(* CoDeSys 2.3.9.41 project: KS Sheksninskaya.pro *)
(* Libraries: PID_Regulators.lib 6.11.19 15:29:27, Util.lib 18.5.10 15:14:28, Germes_1_0.lib 3.5.20 13:44:14, STANDARD.LIB 4.10.05 11:14:46, IECSFC.LIB 13.4.06 15:51:28, SYSLIBTIME.LIB 6.11.19 15:29:28, ANALYZATION.LIB 5.10.99 09:05:06 *)

(* PLC configuration (modules and I/O channels)
Fast discrete inputs [I_SIMPLE_INPUT] node 0, in %IB0 out %QB0 {Filtrationtime = 10}
  DD2_7_DI0 AT %IX0.0 [BitInput] Импульсный счетчик FQS03.01
  DD2_7_DI1 AT %IX0.1 [BitInput] резерв
  DD2_7_DI2 AT %IX0.2 [BitInput] резерв
  DD2_7_DI3 AT %IX0.3 [BitInput] резерв
Discrete inputs [ID130] node 1, in %IB1 out %QB1 {Filtrationtime_GeneralINP = 10; Visibility = No; PinCount = 12}
  AT %IB1.0 [ByteInput] 8 discrete inputs
  AT %IB1.1 [ByteInput] 4 discrete inputs
Discrete outputs [ID131] node 2, in %IB2 out %QB2 {SafeValueByte = 0; SafeValueByteM = 0; Visibility = No; PinCount = 12}
  AT %QB2.0 [ByteOutput] 8 discrete outputs
  AT %QB2.1 [ByteOutput] 4 discrete outputs
Fast analog inputs [ID125] node 3, in %IB3 out %QB3 {Flt_Comm = 50Hz 2Por}
  DD2_7_AI0 AT %IR3.0 [FloatInputP] Датчик температуры в помещении {AIN_TYPE = 0-20 mA; Peak_Filtr = 200; Flt_Ch = Off; TauRC = 10; MinFV = 0; MaxFV = 20}
  DD2_7_AI1 AT %IR3.1 [FloatInputP] Расходомер FT01.01 {AIN_TYPE = 0-20 mA; Peak_Filtr = 200; Flt_Ch = Off; TauRC = 10; MinFV = 0; MaxFV = 20}
  DD2_7_AI2 AT %IR3.2 [FloatInputP] Расходомер FT01.02 {AIN_TYPE = 0-20 mA; Peak_Filtr = 200; Flt_Ch = Off; TauRC = 10; MinFV = 0; MaxFV = 20}
  DD2_7_AI3 AT %IR3.3 [FloatInputP] рН/ОВП метр QE01.01 {AIN_TYPE = 0-20 mA; Peak_Filtr = 200; Flt_Ch = Off; TauRC = 10; MinFV = 0; MaxFV = 20}
  DD2_7_AI4 AT %IR3.4 [FloatInputP] рН/ОВП метр QE01.02 {AIN_TYPE = 0-20 mA; Peak_Filtr = 200; Flt_Ch = Off; TauRC = 10; MinFV = 0; MaxFV = 20}
  DD2_7_AI5 AT %IR3.5 [FloatInputP] Давление на входе в фильтр-пресс {AIN_TYPE = 0-20 mA; Peak_Filtr = 200; Flt_Ch = Off; TauRC = 10; MinFV = 0; MaxFV = 20}
  DD2_7_AI6 AT %IR3.6 [FloatInputP] резерв {AIN_TYPE = 0-20 mA; Peak_Filtr = 200; Flt_Ch = Off; TauRC = 10; MinFV = 0; MaxFV = 20}
  DD2_7_AI7 AT %IR3.7 [FloatInputP] резерв {AIN_TYPE = 0-20 mA; Peak_Filtr = 200; Flt_Ch = Off; TauRC = 10; MinFV = 0; MaxFV = 20}
  AT %IW3.8 [WordInput] AI read time (10ms)
Analog outputs [ID126] node 4, in %IB4 out %QB4
  DD2_7_AO0 AT %QR4.0 [FloatOutputP] Управление НД08.04 {AOUT_TYPE = 4-20 mA; SafeValueREAL = 0.0}
  DD2_7_AO1 AT %QR4.1 [FloatOutputP] резерв {AOUT_TYPE = 4-20 mA; SafeValueREAL = 0.0}
  DD2_7_AO2 AT %QR4.2 [FloatOutputP] резерв {AOUT_TYPE = 4-20 mA; SafeValueREAL = 0.0}
  DD2_7_AO3 AT %QR4.3 [FloatOutputP] резерв {AOUT_TYPE = 4-20 mA; SafeValueREAL = 0.0}
Special input [ID103] node 5, in %IB5 out %QB5 {Filtrationtime = 1000; PinCount = 1; WatchDogPeriod = 400; PollPeriod = 3000; Visibility = No}
  AT %IX5.0 [BitInput] Special input
Special output [ID104] node 6, in %IB6 out %QB6 {Visibility = No; PinCount = 1}
  AT %QX6.0 [BitOutput] Special output
ModBus (Master) [MODBUS_MASTER_ID450] node 7, in %IB7 out %QB7 {Visibility = No}
  LastAddress AT %QD7.0 [DWordOutput] Last address
  LastError AT %QW7.1 [WordOutput] Last error
  RS-485-1 [COM1_USART] node 0, in %IB7.0 out %QB7.0 {CommunicationSpeed = 9600; Parity = EVEN; BitLength = 8 bits; StopLength = One stop bit; InterfaceType = RS485; FrameOriented = RTU; Timeout = 0; Visibility = No}
  Universal Modbus device [ID2000] node 1, in %IB7.1 out %QB7.1 {ModuleIP = 10:0:0:101; ServiceTimeout = 20; TCPport = 502; NetMode = Serial; ModuleSlaveAddress = 11; RequestType = Both; PeriodOfService = 100; Visibility = No; RepeatCounter = 0; ByteSequence = Trace_mode}
    AT %QB7.1.0 [ComChannel] Command (0xff - Start)
    32bit output module [ID2006] node 0, in %IB7.1.0 out %QB7.1.0 {ModbusAddress = 0; Command_write_regs = Force multiple coils (0x0f); Visibility = No}
      DD1_1_DO AT %QD7.1.0.0 [DWordOutput]
  Universal Modbus device [ID2000] node 2, in %IB7.2 out %QB7.2 {ModuleIP = 10:0:0:102; ServiceTimeout = 20; TCPport = 502; NetMode = Serial; ModuleSlaveAddress = 12; RequestType = By poll time; PeriodOfService = 100; Visibility = No; RepeatCounter = 0; ByteSequence = Trace_mode}
    AT %QB7.2.0 [ComChannel] Command (0xff - Start)
DD1_2_DI AT %ID7.2.0.0 [DWordInput]
Universal Modbus device [ID2000] node 3, in %IB7.3 out %QB7.3 {ModuleIP = 10:0:0:103; ServiceTimeout = 20; TCPport = 502; NetMode = Serial; ModuleSlaveAddress = 13; RequestType = By poll time; PeriodOfService = 100; Visibility = No; RepeatCounter = 0; ByteSequence = Trace_mode}
  AT %QB7.3.0 [ComChannel] Command (0xff - Start)
DD1_3_DI AT %IW7.3.0.0 [WordInput]
Universal Modbus device [ID2000] node 4, in %IB7.4 out %QB7.4 {ModuleIP = 10:0:0:104; ServiceTimeout = 20; TCPport = 502; NetMode = Serial; ModuleSlaveAddress = 14; RequestType = Both; PeriodOfService = 100; Visibility = No; RepeatCounter = 0; ByteSequence = Trace_mode}
  AT %QB7.4.0 [ComChannel] Command (0xff - Start)
  Register output module [ID2004] node 0, in %IB7.4.0 out %QB7.4.0 {ModbusAddress = 0; Command_write_one_reg = Write multiple registers(0x10); Visibility = No}
    DD1_4_AO0 AT %QW7.4.0.0 [WordOutput]
  Register output module [ID2004] node 1, in %IB7.4.1 out %QB7.4.1 {ModbusAddress = 1; Command_write_one_reg = Write multiple registers(0x10); Visibility = No}
    DD1_4_AO1 AT %QW7.4.1.0 [WordOutput]
  Register output module [ID2004] node 2, in %IB7.4.2 out %QB7.4.2 {ModbusAddress = 2; Command_write_one_reg = Write multiple registers(0x10); Visibility = No}
    DD1_4_AO2 AT %QW7.4.2.0 [WordOutput]
  Register output module [ID2004] node 3, in %IB7.4.3 out %QB7.4.3 {ModbusAddress = 3; Command_write_one_reg = Write multiple registers(0x10); Visibility = No}
    DD1_4_AO3 AT %QW7.4.3.0 [WordOutput]
  Register output module [ID2004] node 4, in %IB7.4.4 out %QB7.4.4 {ModbusAddress = 4; Command_write_one_reg = Write multiple registers(0x10); Visibility = No}
    DD1_4_AO4 AT %QW7.4.4.0 [WordOutput]
  Register output module [ID2004] node 5, in %IB7.4.5 out %QB7.4.5 {ModbusAddress = 5; Command_write_one_reg = Write multiple registers(0x10); Visibility = No}
    DD1_4_AO5 AT %QW7.4.5.0 [WordOutput]
  Register output module [ID2004] node 6, in %IB7.4.6 out %QB7.4.6 {ModbusAddress = 6; Command_write_one_reg = Write multiple registers(0x10); Visibility = No}
    DD1_4_AO6 AT %QW7.4.6.0 [WordOutput]
  Register output module [ID2004] node 7, in %IB7.4.7 out %QB7.4.7 {ModbusAddress = 7; Command_write_one_reg = Write multiple registers(0x10); Visibility = No}
    DD1_4_AO7 AT %QW7.4.7.0 [WordOutput]
  AT %QB7.5.0 [ComChannel] Command (0xff - Start)
com_wordN0105 AT %QW7.5.0.0 [WordOutput]
zad_rsN0105 AT %QW7.5.1.0 [WordOutput]
stat_wordN0105 AT %IW7.5.2.0 [WordInput]
di29N0105 AT %IW7.5.3.0 [WordInput]
Universal Modbus device [ID2000] node 6, in %IB7.6 out %QB7.6 {ModuleIP = 10:0:0:106; ServiceTimeout = 20; TCPport = 502; NetMode = Serial; ModuleSlaveAddress = 16; RequestType = By poll time; PeriodOfService = 100; Visibility = No; RepeatCounter = 0; ByteSequence = Trace_mode}
  AT %QB7.6.0 [ComChannel] Command (0xff - Start)
  Register output module [ID2004] node 0, in %IB7.6.0 out %QB7.6.0 {ModbusAddress = 49999; Command_write_one_reg = Write multiple registers(0x10); Visibility = No}
    com_wordND080301 AT %QW7.6.0.0 [WordOutput]
  Register output module [ID2004] node 1, in %IB7.6.1 out %QB7.6.1 {ModbusAddress = 50009; Command_write_one_reg = Write multiple registers(0x10); Visibility = No}
    zad_rsND080301 AT %QW7.6.1.0 [WordOutput]
  Register input module [ID2003] node 2, in %IB7.6.2 out %QB7.6.2 {ModbusAddress = 50199; Command_read_regs = Read holding Registers  (0x03); Visibility = No}
    stat_wordND080301 AT %IW7.6.2.0 [WordInput]
  Register input module [ID2003] node 3, in %IB7.6.3 out %QB7.6.3 {ModbusAddress = 16609; Command_read_regs = Read holding Registers  (0x03); Visibility = No}
    di29ND080301 AT %IW7.6.3.0 [WordInput]
Universal Modbus device [ID2000] node 7, in %IB7.7 out %QB7.7 {ModuleIP = 10:0:0:107; ServiceTimeout = 20; TCPport = 502; NetMode = Serial; ModuleSlaveAddress = 17; RequestType = By poll time; PeriodOfService = 100; Visibility = No; RepeatCounter = 0; ByteSequence = Trace_mode}
  AT %QB7.7.0 [ComChannel] Command (0xff - Start)
com_wordND080302 AT %QW7.7.0.0 [WordOutput]
zad_rsND080302 AT %QW7.7.1.0 [WordOutput]
stat_wordND080302 AT %IW7.7.2.0 [WordInput]
di29ND080302 AT %IW7.7.3.0 [WordInput]
Universal Modbus device [ID2000] node 8, in %IB7.8 out %QB7.8 {ModuleIP = 10:0:0:201; ServiceTimeout = 20; TCPport = 502; NetMode = Serial; ModuleSlaveAddress = 21; RequestType = Both; PeriodOfService = 100; Visibility = No; RepeatCounter = 0; ByteSequence = Trace_mode}
  AT %QB7.8.0 [ComChannel] Command (0xff - Start)
  32bit output module [ID2006] node 0, in %IB7.8.0 out %QB7.8.0 {ModbusAddress = 0; Command_write_regs = Force multiple coils (0x0f); Visibility = No}
    DD2_1_DO AT %QD7.8.0.0 [DWordOutput]
Universal Modbus device [ID2000] node 9, in %IB7.9 out %QB7.9 {ModuleIP = 10:0:0:202; ServiceTimeout = 20; TCPport = 502; NetMode = Serial; ModuleSlaveAddress = 22; RequestType = Both; PeriodOfService = 100; Visibility = No; RepeatCounter = 0; ByteSequence = Trace_mode}
  AT %QB7.9.0 [ComChannel] Command (0xff - Start)
DD2_2_DO AT %QD7.9.0.0 [DWordOutput]
Universal Modbus device [ID2000] node 10, in %IB7.10 out %QB7.10 {ModuleIP = 10:0:0:203; ServiceTimeout = 20; TCPport = 502; NetMode = Serial; ModuleSlaveAddress = 23; RequestType = Both; PeriodOfService = 100; Visibility = No; RepeatCounter = 0; ByteSequence = Trace_mode}
  AT %QB7.10.0 [ComChannel] Command (0xff - Start)
DD2_3_DO AT %QW7.10.0.0 [WordOutput]
Universal Modbus device [ID2000] node 11, in %IB7.11 out %QB7.11 {ModuleIP = 10:0:0:204; ServiceTimeout = 20; TCPport = 502; NetMode = Serial; ModuleSlaveAddress = 24; RequestType = By poll time; PeriodOfService = 100; Visibility = No; RepeatCounter = 0; ByteSequence = Trace_mode}
  AT %QB7.11.0 [ComChannel] Command (0xff - Start)
DD2_4_DI AT %ID7.11.0.0 [DWordInput]
Universal Modbus device [ID2000] node 12, in %IB7.12 out %QB7.12 {ModuleIP = 10:0:0:205; ServiceTimeout = 20; TCPport = 502; NetMode = Serial; ModuleSlaveAddress = 25; RequestType = By poll time; PeriodOfService = 100; Visibility = No; RepeatCounter = 0; ByteSequence = Trace_mode}
  AT %QB7.12.0 [ComChannel] Command (0xff - Start)
DD2_5_DI AT %ID7.12.0.0 [DWordInput]
Universal Modbus device [ID2000] node 13, in %IB7.13 out %QB7.13 {ModuleIP = 10:0:0:206; ServiceTimeout = 20; TCPport = 502; NetMode = Serial; ModuleSlaveAddress = 26; RequestType = By poll time; PeriodOfService = 100; Visibility = No; RepeatCounter = 0; ByteSequence = Trace_mode}
  AT %QB7.13.0 [ComChannel] Command (0xff - Start)
DD2_6_DI AT %ID7.13.0.0 [DWordInput]
Universal Modbus device [ID2000] node 14, in %IB7.14 out %QB7.14 {ModuleIP = 10:0:0:301; ServiceTimeout = 20; TCPport = 502; NetMode = Serial; ModuleSlaveAddress = 31; RequestType = Both; PeriodOfService = 100; Visibility = No; RepeatCounter = 0; ByteSequence = Trace_mode}
  AT %QB7.14.0 [ComChannel] Command (0xff - Start)
  8 bit output module [ID2002] node 0, in %IB7.14.0 out %QB7.14.0 {ModbusAddress = 241; Command_write_byte = Force multiply coils (0x0f); Visibility = No}
    AT %QB7.14.0.0 [ByteOutput]
  8 bit input module [ID2001] node 1, in %IB7.14.1 out %QB7.14.1 {ModbusAddress = 201; Command_read_byte = Read coils status (0x01); Visibility = No}
    AT %IB7.14.1.0 [ByteInput]
Universal Modbus device [ID2000] node 15, in %IB7.15 out %QB7.15 {ModuleIP = 10:0:0:302; ServiceTimeout = 20; TCPport = 502; NetMode = Serial; ModuleSlaveAddress = 32; RequestType = Both; PeriodOfService = 100; Visibility = No; RepeatCounter = 0; ByteSequence = Trace_mode}
  AT %QB7.15.0 [ComChannel] Command (0xff - Start)
  8 bit output module [ID2002] node 0, in %IB7.15.0 out %QB7.15.0 {ModbusAddress = 241; Command_write_byte = Force multiply coils (0x0f); Visibility = No}
    AT %QB7.15.0.0 [ByteOutput]
  8 bit input module [ID2001] node 1, in %IB7.15.1 out %QB7.15.1 {ModbusAddress = 201; Command_read_byte = Read coils status (0x01); Visibility = No}
    AT %IB7.15.1.0 [ByteInput]
AT %QD8.0 [DWordOutput] Last address
AT %QW8.1 [WordOutput] Last error
RS-232 [COM2_USART] node 0, in %IB8.0 out %QB8.0 {CommunicationSpeed = 11520; Parity = NO PARITY CHECK; BitLength = 8 bits; StopLength = One stop bit; InterfaceType = RS232; FrameOriented = RTU; Timeout = 0; Visibility = No}
AT %QB8.1.0 [ComChannel] Command (0xff - Start)
valueTemperaturePAN AT %QD8.1.0.0 [FloatOutput]
valueFT0101PAN AT %QD8.1.1.0 [FloatOutput]
valueFT0102PAN AT %QD8.1.2.0 [FloatOutput]
valueQE0101PAN AT %QD8.1.3.0 [FloatOutput]
valueQE0102PAN AT %QD8.1.4.0 [FloatOutput]
valueFPKpressurePAN AT %QD8.1.5.0 [FloatOutput]
totalAmountFQS0301PAN AT %QD8.1.6.0 [FloatOutput]
toNextRegenPAN AT %QD8.1.7.0 [FloatOutput]
counterND050201PAN AT %QD8.1.8.0 [FloatOutput]
counterND050202PAN AT %QD8.1.9.0 [FloatOutput]
daysND050201PAN AT %QW8.1.10.0 [WordOutput]
hoursND050201PAN AT %QW8.1.11.0 [WordOutput]
minutesND050201PAN AT %QW8.1.12.0 [WordOutput]
secondsND050201PAN AT %QW8.1.13.0 [WordOutput]
daysND050202PAN AT %QW8.1.14.0 [WordOutput]
hoursND050202PAN AT %QW8.1.15.0 [WordOutput]
minutesND050202PAN AT %QW8.1.16.0 [WordOutput]
secondsND050202PAN AT %QW8.1.17.0 [WordOutput]
counterND060201PAN AT %QD8.1.18.0 [FloatOutput]
counterND060202PAN AT %QD8.1.19.0 [FloatOutput]
daysND060201PAN AT %QW8.1.20.0 [WordOutput]
hoursND060201PAN AT %QW8.1.21.0 [WordOutput]
minutesND060201PAN AT %QW8.1.22.0 [WordOutput]
secondsND060201PAN AT %QW8.1.23.0 [WordOutput]
daysND060202PAN AT %QW8.1.24.0 [WordOutput]
hoursND060202PAN AT %QW8.1.25.0 [WordOutput]
minutesND060202PAN AT %QW8.1.26.0 [WordOutput]
secondsND060202PAN AT %QW8.1.27.0 [WordOutput]
counterND060301PAN AT %QD8.1.28.0 [FloatOutput]
counterND060302PAN AT %QD8.1.29.0 [FloatOutput]
daysND060301PAN AT %QW8.1.30.0 [WordOutput]
hoursND060301PAN AT %QW8.1.31.0 [WordOutput]
minutesND060301PAN AT %QW8.1.32.0 [WordOutput]
secondsND060301PAN AT %QW8.1.33.0 [WordOutput]
daysND060302PAN AT %QW8.1.34.0 [WordOutput]
hoursND060302PAN AT %QW8.1.35.0 [WordOutput]
minutesND060302PAN AT %QW8.1.36.0 [WordOutput]
secondsND060302PAN AT %QW8.1.37.0 [WordOutput]
counterND070301PAN AT %QD8.1.38.0 [FloatOutput]
counterND070302PAN AT %QD8.1.39.0 [FloatOutput]
daysND070301PAN AT %QW8.1.40.0 [WordOutput]
hoursND070301PAN AT %QW8.1.41.0 [WordOutput]
minutesND070301PAN AT %QW8.1.42.0 [WordOutput]
secondsND070301PAN AT %QW8.1.43.0 [WordOutput]
daysND070302PAN AT %QW8.1.44.0 [WordOutput]
hoursND070302PAN AT %QW8.1.45.0 [WordOutput]
minutesND070302PAN AT %QW8.1.46.0 [WordOutput]
secondsND070302PAN AT %QW8.1.47.0 [WordOutput]
counterND080301PAN AT %QD8.1.48.0 [FloatOutput]
counterND080302PAN AT %QD8.1.49.0 [FloatOutput]
daysND080301PAN AT %QW8.1.50.0 [WordOutput]
hoursND080301PAN AT %QW8.1.51.0 [WordOutput]
minutesND080301PAN AT %QW8.1.52.0 [WordOutput]
secondsND080301PAN AT %QW8.1.53.0 [WordOutput]
daysND080302PAN AT %QW8.1.54.0 [WordOutput]
hoursND080302PAN AT %QW8.1.55.0 [WordOutput]
minutesND080302PAN AT %QW8.1.56.0 [WordOutput]
secondsND080302PAN AT %QW8.1.57.0 [WordOutput]
counterN010501PAN AT %QD8.1.58.0 [FloatOutput]
counterN010502PAN AT %QD8.1.59.0 [FloatOutput]
daysN010501PAN AT %QW8.1.60.0 [WordOutput]
hoursN010501PAN AT %QW8.1.61.0 [WordOutput]
minutesN010501PAN AT %QW8.1.62.0 [WordOutput]
secondsN010501PAN AT %QW8.1.63.0 [WordOutput]
daysN010502PAN AT %QW8.1.64.0 [WordOutput]
hoursN010502PAN AT %QW8.1.65.0 [WordOutput]
minutesN010502PAN AT %QW8.1.66.0 [WordOutput]
secondsN010502PAN AT %QW8.1.67.0 [WordOutput]
counterN040401PAN AT %QD8.1.68.0 [FloatOutput]
counterN040402PAN AT %QD8.1.69.0 [FloatOutput]
daysN040401PAN AT %QW8.1.70.0 [WordOutput]
hoursN040401PAN AT %QW8.1.71.0 [WordOutput]
minutesN040401PAN AT %QW8.1.72.0 [WordOutput]
secondsN040401PAN AT %QW8.1.73.0 [WordOutput]
daysN040402PAN AT %QW8.1.74.0 [WordOutput]
hoursN040402PAN AT %QW8.1.75.0 [WordOutput]
minutesN040402PAN AT %QW8.1.76.0 [WordOutput]
secondsN040402PAN AT %QW8.1.77.0 [WordOutput]
counterUFO030101PAN AT %QD8.1.78.0 [FloatOutput]
counterUFO030102PAN AT %QD8.1.79.0 [FloatOutput]
daysUFO030101PAN AT %QW8.1.80.0 [WordOutput]
hoursUFO030101PAN AT %QW8.1.81.0 [WordOutput]
minutesUFO030101PAN AT %QW8.1.82.0 [WordOutput]
secondsUFO030101PAN AT %QW8.1.83.0 [WordOutput]
daysUFO030102PAN AT %QW8.1.84.0 [WordOutput]
hoursUFO030102PAN AT %QW8.1.85.0 [WordOutput]
minutesUFO030102PAN AT %QW8.1.86.0 [WordOutput]
secondsUFO030102PAN AT %QW8.1.87.0 [WordOutput]
counterN020401PAN AT %QD8.1.88.0 [FloatOutput]
counterN020402PAN AT %QD8.1.89.0 [FloatOutput]
daysN020401PAN AT %QW8.1.90.0 [WordOutput]
hoursN020401PAN AT %QW8.1.91.0 [WordOutput]
minutesN020401PAN AT %QW8.1.92.0 [WordOutput]
secondsN020401PAN AT %QW8.1.93.0 [WordOutput]
daysN020402PAN AT %QW8.1.94.0 [WordOutput]
hoursN020402PAN AT %QW8.1.95.0 [WordOutput]
minutesN020402PAN AT %QW8.1.96.0 [WordOutput]
secondsN020402PAN AT %QW8.1.97.0 [WordOutput]
statusNDstartPAN AT %QW8.1.98.0 [WordOutput]
statusStartPAN AT %QW8.1.99.0 [WordOutput]
valveOpenedPAN AT %QD8.1.100.0 [DWordOutput]
regimeFSPAN AT %QW8.1.101.0 [WordOutput]
levelStatusPAN AT %QW8.1.102.0 [WordOutput]
valveClosedPAN AT %QD8.1.103.0 [DWordOutput]
statWordND0502PAN AT %QW8.1.104.0 [WordOutput]
statWordND0602PAN AT %QW8.1.105.0 [WordOutput]
statWordND0603PAN AT %QW8.1.106.0 [WordOutput]
statWordND0703PAN AT %QW8.1.107.0 [WordOutput]
statWordND0803PAN AT %QW8.1.108.0 [WordOutput]
statWordN0105PAN AT %QW8.1.109.0 [WordOutput]
statWordN0404PAN AT %QW8.1.110.0 [WordOutput]
statWordUFO0301PAN AT %QW8.1.111.0 [WordOutput]
statWordN0204PAN AT %QW8.1.112.0 [WordOutput]
alarmAIPAN AT %QW8.1.113.0 [WordOutput]
alarmToOpenValvePAN AT %QD8.1.114.0 [DWordOutput]
alarmToCloseValvePAN AT %QD8.1.115.0 [DWordOutput]
alarmFSPAN AT %QW8.1.116.0 [WordOutput]
failToRegenFSPAN AT %QW8.1.117.0 [WordOutput]
AT %QB8.1.118.0 [ByteOutput]
AT %QB8.1.119.0 [ByteOutput]
Universal Modbus device [ID2000] node 2, in %IB8.2 out %QB8.2 {ModuleIP = 10:0:0:223; ServiceTimeout = 150; TCPport = 502; NetMode = Serial; ModuleSlaveAddress = 1; RequestType = By poll time; PeriodOfService = 10; Visibility = No; RepeatCounter = 0; ByteSequence = Native}
  AT %QB8.2.0 [ComChannel] Command (0xff - Start)
impulsValueFQS0301PAN AT %ID8.2.0.0 [FloatInput]
timeToWorkFPKPAN AT %IW8.2.1.0 [WordInput]
maxPressureValueFPKPAN AT %IW8.2.2.0 [WordInput]
ND0502setMaxDosValPAN AT %ID8.2.3.0 [FloatInput]
ND0502setKoefPropPAN AT %ID8.2.4.0 [FloatInput]
ND0602setMaxDosValPAN AT %ID8.2.5.0 [FloatInput]
ND0602setKoefPropPAN AT %ID8.2.6.0 [FloatInput]
ND0603setMaxDosValPAN AT %ID8.2.7.0 [FloatInput]
ND0603setKoefPropPAN AT %ID8.2.8.0 [FloatInput]
ND0703pHsetValuePAN AT %ID8.2.9.0 [FloatInput]
ND0703YoutManualPAN AT %ID8.2.10.0 [FloatInput]
ND0803setMaxDosValPAN AT %ID8.2.11.0 [FloatInput]
ND0803setKoefPropPAN AT %ID8.2.12.0 [FloatInput]
ND0804doseValuePAN AT %ID8.2.13.0 [FloatInput]
N0105flowSetValuePAN AT %ID8.2.14.0 [FloatInput]
N0105YoutManualPAN AT %ID8.2.15.0 [FloatInput]
setVolumeFSPAN AT %ID8.2.16.0 [FloatInput]
setMinTemperaturePAN AT %ID8.2.17.0 [FloatInput]
setMaxTemperaturePAN AT %ID8.2.18.0 [FloatInput]
correctionValueFQS0301PAN AT %ID8.2.19.0 [FloatInput]
setWordND0502PAN AT %IW8.2.20.0 [WordInput]
setWordND0602PAN AT %IW8.2.21.0 [WordInput]
setWordND0603PAN AT %IW8.2.22.0 [WordInput]
setWordND0703PAN AT %IW8.2.23.0 [WordInput]
setWordND0803PAN AT %IW8.2.24.0 [WordInput]
setWordN0105PAN AT %IW8.2.25.0 [WordInput]
setWordN0404PAN AT %IW8.2.26.0 [WordInput]
setWordUFO0301PAN AT %IW8.2.27.0 [WordInput]
setWordN0204PAN AT %IW8.2.28.0 [WordInput]
%MtestValvePAN AT %ID8.2.29.0 [DWordInput]
AT %IB8.2.30.0 [ByteInput]
AT %IB8.2.31.0 [ByteInput]
ModBus (slave) [MODBUS_ID400] node 9, in %IB9 out %QB9 {SlaveIdentificator = 1; Visibility = No}
TCP [TCP_ID221] node 0, in %IB9.0.0 out %QB9.0.0 {RemotePort = 502; Visibility = No}
remFT0101value AT %QD9.1.0 [FloatOutput]
remFQS0301totalAmount AT %QD9.2.0 [FloatOutput]
remTemperatureValue AT %QD9.3.0 [FloatOutput]
AT %QB9.4.0 [ByteOutput]
AT %QB9.5.0 [ByteOutput]
*)

(* POU PLC_PRG, CFC *)
PROGRAM PLC_PRG
VAR
	alarm: BOOL; (*Общий сигнал авария *)
	resetAlarms: BOOL;		(*Сброс аварий.*)
	ControlAI0: ControlAI;		(*Блок контроля входа AI1 ПЛК.*)
	ControlAI1: ControlAI;		(*Блок контроля входа AI2 ПЛК.*)
	ControlAI2: ControlAI;		(*Блок контроля входа AI3 ПЛК.*)
	ControlAI3: ControlAI;		(*Блок контроля входа AI4 ПЛК.*)
	ControlAI4: ControlAI;		(*Блок контроля входа AI5 ПЛК.*)
	ControlAI5: ControlAI;		(*Блок контроля входа AI6 ПЛК.*)
	valueTemperature: REAL;		(*Температура в помещении*)
	valueFT0101: REAL;		(*Показания расходомера на входе в станцию.*)
	valueFT0102: REAL;		(*Показания расходомера после отстойника.*)
	valueQE0101: REAL;		(*Показания рН-метра на входе в станцию.*)
	valueQE0102: REAL;		(*Показания рН-метра после отстойника.*)
	valueFPKpressure: REAL;		(*Давление на входе в фильтр-пресс.*)
	alarmAI: WORD;		(*0 - Авария датчика температуры.
							1 - Авария расходомера FT01.01.
							2 - Авария расходомера FT01.02.
							3 - Авария рН-метра QE01.01.
							4 - Авария рН-метра QE01.02.
							5 - Авария входа приема показаний давления на входе в фильтр.*)
	setMinTemperature: REAL;		(*Задать минимальную температуру.*)
	setMaxTemperature: REAL;		(*Задать максимальную температуру.*)
	alarmTemperatureHigh: BOOL;		(*Авария - температура в помещении выше заданного максимального значения.*)
	alarmTemperatureLow: BOOL;		(*Авария - температура в помещении ниже заданного минимального значения.*)
	CounterFQS0301impulses: ImpulsFlowCounter;		(*Счетчик очищенных стоков.*)
	impulsValueFQS0301: REAL;		(*Вес импульса расходомера.*)
	resetCounterFQS0301: BOOL;		(*Сброс счетчика QS03.01*)
	correctionValueFQS0301: REAL;		(*Величина коррекции счетчика.*)
	addCorrectionFQS0301: BOOL;		(*Прибавить величину коррекции к текущему значению счетчика.*)
	deleteCorrectionFQS0301: BOOL;		(*Вычесть величину коррекции из текущего значения счетчика.*)
	alarmND: WORD;		(*Сигнал авария от насосов дозаторов.*)
	StartInitiBlock: R_TRIG;		(*Детектор переднего фронта для инициализации требуемых булевых переменных при включении.*)
	startInitializer: BOOL;		(*Переменная для инициализации требуемых булевых переменных при включении.*)
	ND0502dosing: DosingPumpProportional;		(*Блок управления подачей реагента пропорционально расходу.*)
	ND0502manager: RichTwoPumpManager;		(*Блок управления доз.насосами НД05.02.*)
	ND0502setMaxDosVal: REAL;		(*Указать максимальную производительность доз.насоса, мл/мин*)
	ND0502setKoefProp: REAL;		(*Задать количество реагента в мл на один кубометр стоков, мл/м3.*)
	setWordND0502: WORD;		(*Командное слово для управления доз.насосами НД05.02.*)
	statWordND0502: WORD;		(*Слово состояния НД05.02*)
	ND0602dosing: DosingPumpProportional;		(*Блок управления подачей реагента пропорционально расходу.*)
	ND0602manager: RichTwoPumpManager;		(*Блок управления доз.насосами НД06.02.*)
	ND0602setMaxDosVal: REAL;		(*Указать максимальную производительность доз.насоса, мл/мин*)
	ND0602setKoefProp: REAL;		(*Задать количество реагента в мл на один кубометр стоков, мл/м3.*)
	setWordND0602: WORD;		(*Командное слово для управления доз.насосами НД06.02.*)
	statWordND0602: WORD;		(*Слово состояния НД06.02*)
	ND0603dosing: DosingPumpProportional;		(*Блок управления подачей реагента пропорционально расходу.*)
	ND0603manager: RichTwoPumpManager;		(*Блок управления доз.насосами НД06.03.*)
	ND0603setMaxDosVal: REAL;		(*Указать максимальную производительность доз.насоса, мл/мин*)
	ND0603setKoefProp: REAL;		(*Задать количество реагента в мл на один кубометр стоков, мл/м3.*)
	setWordND0603: WORD;		(*Командное слово для управления доз.насосами НД06.03.*)
	statWordND0603: WORD;		(*Слово состояния НД06.03.*)
	ND0703pidReg: PID;		(*Блок ПИД регулирования НД07.03.*)
	ND0703pHsetValue: REAL;		(*Задание рН для поддержания подачей щелочи от НД07.03 по рН метру QE01.01.*)
	ND0703YoutManual: WORD;		(*Ручное задание выходу Y. Задается: 0...100%, на выходе: 4…20мА*)
	manYoutND0703: LIN_TRAFO;		(*Блок преобразования 0...100 в 4...20 для ручного управления выходом ПИД-регулятора.*)
	ND0703manager: RichTwoPumpManager;		(*Блок управления доз.насосами НД07.03.*)
	ND0703YmanAuto: BOOL;		(*Выбор управления выходом Y в ручном или автоматическом режиме.
0 = авто, 1 = ручной*)
	setWordND0703: WORD;		(*Командное слово для управления доз.насосами НД07.03.*)
	statWordND0703: WORD;		(*Слово состояния НД07.03.*)
	ND0803dosing: DosingPumpProportional;		(*Блок управления подачей реагента пропорционально расходу.*)
	ND0803setMaxDosVal: REAL;		(*Указать максимальную производительность доз.насоса, мл/мин*)
	ND0803setKoefProp: REAL;		(*Задать количество реагента в мл на один кубометр стоков, мл/м3.*)
	ND0803manager: RichTwoPumpManager;		(*Блок управления доз.насосами НД08.03.*)
	setWordND0803: WORD;		(*Командное слово для управления доз.насосами НД08.03.*)
	statWordND0803: WORD;		(*Слово состояния НД08.03.*)
	linTrafoND0803: LIN_TRAFO;		(*Блок преобразования сигнала 4...20 в сигнал 0...16384 для ЧРП.*)
	startStopND080301: StartStopVFD;		(*Командное слово в ЧРП НД08.03/01*)
	startStopND080302: StartStopVFD;		(*Командное слово в ЧРП НД08.03/02*)
	linTrafND0804: LIN_TRAFO;		(*Блок преобразования 0...100 в 4...20мА НД08.04*)
	ND0804doseValue: WORD;		(*Задание на дозирование НД08.04 в процентах от максимальной
производительности насоса (0-100), преобразуется пропорционально в сигнал 4…20мА.*)
	PID_ND0105: PID;		(*Блок регулирования производительности Н01.05 для поддержания заданного расхода.*)
	StartStopND0105: StartStopVFD;		(*Блок для запуска и останова ЧРП Н01.05 командным словом по модбасу.*)
	ND0105manager: TwoPumpOneDriveManager;		(*Блок управлением насосами Н01.05*)
	N0105flowSetValue: REAL;		(*Задание расхода для поддержания по FT01.02*)
	N0105YoutManual: WORD;		(*Ручное задание выходу Y. Задается: 0...100%, на выходе: 4…20мА*)
	N0105YmanAuto: BOOL;		(*Выбор управления выходом Y в ручном или автоматическом режиме.
0 = авто, 1 = ручной*)
	linTrafoN0105: LIN_TRAFO;		(*Блок преобразования 0...100 в 0...16384 для ручного управления выходом ПИД-регулятора.*)
	rsTrigN0105: RS;		(*Защелка сигнала на пуск насосов Н01.05*)
	N0105manStart: BOOL;		(*Ручной пуск Н01.05*)
	N0105manStop: BOOL;		(*Ручной стоп Н01.05*)
	setWordN0105: WORD;		(*Командное слово для управления доз.насосами Н01.05*)
	statWordN0105: WORD;		(*Слово состояния Н01.05*)
	setRegimeFS: WORD;		(*Подача управляющего сигнала в клапан фильтра.
0=нет сигнала, 1 = начать промывку.*)
	regimeFS: WORD;		(*Сигнал от управляющего клапана фильтра о текущем режиме:
0 = фильтрация, 1 = промывка.*)
	alarmFS: WORD;		(*Сигнал авария от управляющего клапана фильтра.
0 = авария, 1 = промывка.*)
	regeneratedFS: WORD; (*1 = статус - регенерация проведена*)
	failToRegenFS: WORD; (*1 = регенерация не удалась.*)
	openedKEM: WORD;		(*Статус - клапан КЭМ открыт.*)
	openValve: DWORD;		(*Сигнал на открытие заслонки*)
	closeValve: DWORD;		(*Сигнал на закрытие заслонки*)
	valveOpened: DWORD;		(*Статус - заслонка ОТКРЫТА*)
	valveClosed: DWORD;		(*Статус - заслонка ЗАКРЫТА*)
	alarmToOpenValve: DWORD;		(*Авария на открытие (заслонка не открылась за заданное время)*)
	alarmToCloseValve: DWORD;		(*Авария на закрытие (заслонка не закрылась за заданное время)*)
	testValve: DWORD; (*Тестировать заслонку. 1 = открыть, 0 = закрыть.*)
	N0204manager: RichTwoPumpManager;		(*Блок управления насосами Н02.04*)
	N0204manStart: BOOL;		(*Ручной пуск Н02.04*)
	N0204manStop: BOOL;		(*Ручной стоп Н02.04*)
	N0204startTrig: RS;		(*Триггер ручного пуска/останова насоса Н02.04*)
	setWordN0204: WORD;		(*Командное слово для управления доз.насосами Н02.04*)
	statWordN0204: WORD;		(*Слово состояния насосов Н02.04*)
	N0404manager: RichTwoPumpManager;		(*Блок управления дренажными насосами Н04.04*)
	N0404manStart: BOOL;		(*Ручной пуск Н04.04*)
	N0404manStop: BOOL;		(*Ручной стоп Н04.04*)
	N0404startTrig: RS;		(*Триггер ручного пуск/стоп насосов Н04.04*)
	setWordN0404: WORD;		(*Командное слово управления насосами Н04.04*)
	statWordN0404: WORD;		(*Слово состояния насосов Н04.04*)
	timeToWorkFPK: WORD := 900;		(*Время работы ФПК после спада сигнала уровня осадка, сек.
по умолчанию 15 мин.*)
	FPKstopTimer: TOF;		(*Таймер задержки снятия сигнала на выключение ФПК после спада сигнала уровня осадка.*)
	FPKstopFtrig: F_TRIG;		(*Детектор спада сигнала уровня осадка после таймера на отключение.*)
	FPKstartTrig: RS;		(*Триггер сигнала на пуск/стоп фильтр-пресса.*)
	maxPressureValueFPK: WORD := 10;		(*Максимально допустимое давление на входе ФПК, 0...16 бар.
			По умолчанию 10.*)
	needToCleanFPK: BOOL;		(*Сигнал о необходимости почистить фильтр-пресс.*)
	needToClleanFPKtrig: RS;		(*Триггер контроля сигнала о необходимости почистить фильтр-пресс.*)
	readyFPKrTrig: R_TRIG;		(*Детектор появления сигнала о готовности фильтр-пресса к работе.*)
	notStartedFPKtimer: TON;		(*Таймер контроля запуска ФПК.*)
	notStartedFPK: BOOL;		(*Фильтр-пресс не запустился через 5 мин после подачи сигнала на запуск.*)
	valveKSHE0401: SimpleValve;		(*Блок управления заслонкой КШЭ04.01*)
	valveZDE0225: SimpleValve;		(*Блок управления заслонкой наполнения РЧВ = ЗДЭ02.25*)
	regenByFT0102: FlowVolume;		(*Блок подачи сигнала на промывку после прохождения заданного объема по FT01.02.*)
	FS020101: QueueManager;		(*Блок управления ФС02.01/01*)
	FS020102: QueueManager;		(*Блок управления ФС02.01/02*)
	FS020103: QueueManager;		(*Блок управления ФС02.01/03*)
	FS020104: QueueManager;		(*Блок управления ФС02.01/04*)
	FS020105: QueueManager;		(*Блок управления ФС02.01/05*)
	FS020106: QueueManager;		(*Блок управления ФС02.01/06*)
	FS020201: QueueManager;		(*Блок управления ФС02.02/01*)
	FS020202: QueueManager;		(*Блок управления ФС02.02/02*)
	FS020203: QueueManager;		(*Блок управления ФС02.02/03*)
	FS020204: QueueManager;		(*Блок управления ФС02.02/04*)
	FS020205: QueueManager;		(*Блок управления ФС02.02/05*)
	FS020206: QueueManager;		(*Блок управления ФС02.02/06*)
	totalAmountFS: REAL;		(*Сумма стоков прошедших через счетчик FS01.02 на фильтрацию, кубометров*)
	setVolumeFS: REAL;		(*Задание объема до следующей промывки, кубометров.*)
	resetVolumeFS: BOOL;		(*Сброс счетчика до промывки*)
	UFO0301manager: RichTwoPumpManager;		(*Блок управления УФО03.01*)
	ZDE0301: SimpleValve;		(*Блок управления задвижкой ЗДЭ03.01 для УФО03.01/01*)
	ZDE0302: SimpleValve;		(*Блок управления задвижкой ЗДЭ03.02 для УФО03.01/02*)
	setWordUFO0301: WORD;		(*Командное слово управления УФО03.01*)
	statWordUFO0301: WORD;		(*Слово состояния УФО03.01*)
	ZDE0101: SimpleValve;		(*Блок управления заслонкой ЗДЭ01.01 на входе в станцию.*)
	alarmPLKnetworkDelay: TOF;		(*Задержка выдачи сигнала об обрыве в сети ПЛК.*)
	statusNDstart: WORD;		(*Статус старт насоса дозатора*)
	StatusStart: WORD;		(*Статус старт оборудования*)
	levelStatus: WORD;		(*Статус от сигнализаторов уровня*)
	readyFPK: BOOL;
	powerAlarmN0105: BOOL;
	alarmPLKnetwork: BOOL;
	alarmFPK: BOOL;
	alarmM0604: BOOL;
	alarmM0702: BOOL;
	alarmM0802: BOOL;
	powerAlarmFS: BOOL;
	powerAlarmKEM: BOOL;
	powerAlarmRelay1: BOOL;
	powerAlarmRelay2: BOOL;
	toNextRegen: REAL;		(*Осталось кубометров до следующей промывки*)
	openRS0: RS;
	openRS1: RS;
	openRS2: RS;
	openRS3: RS;
	openRS4: RS;
	openRS5: RS;
	openRS6: RS;
	openRS7: RS;
	openRS8: RS;
	openRS9: RS;
	openRS10: RS;
	openRS11: RS;
	openRS12: RS;
	openRS13: RS;
	openRS14: RS;
	openRS15: RS;
	openRS16: RS;
	openRS17: RS;
	openRS18: RS;
	openRS19: RS;
	openRS20: RS;
	openRS21: RS;
	openRS22: RS;
	openRS23: RS;
	openRS24: RS;
	openRS25: RS;
	openRS26: RS;
	openRS27: RS;
	openRS28: RS;
	closeRS0: RS;
	closeRS1: RS;
	closeRS2: RS;
	closeRS3: RS;
	closeRS4: RS;
	closeRS5: RS;
	closeRS6: RS;
	closeRS7: RS;
	closeRS8: RS;
	closeRS9: RS;
	closeRS10: RS;
	closeRS11: RS;
	closeRS12: RS;
	closeRS13: RS;
	closeRS14: RS;
	closeRS15: RS;
	closeRS16: RS;
	closeRS17: RS;
	closeRS18: RS;
	closeRS19: RS;
	closeRS20: RS;
	closeRS21: RS;
	closeRS22: RS;
	closeRS23: RS;
	closeRS24: RS;
	closeRS25: RS;
	closeRS26: RS;
	closeRS27: RS;
	closeRS28: RS;
	lintrafoND050201: LIN_TRAFO;
	lintrafoND050202: LIN_TRAFO;
	lintrafoND060201: LIN_TRAFO;
	lintrafoND060202: LIN_TRAFO;
	linrtafoND060301: LIN_TRAFO;
	linrtafoND060302: LIN_TRAFO;
	lintrafoND070301: LIN_TRAFO;
	lintrafoND070302: LIN_TRAFO;
END_VAR
VAR RETAIN
	totalAmountFQS0301: DWORD;		(*Итоговая сумма очищенных стоков, выходящих из станции.*)
	counterND050201: DWORD;		(*Счетчик включений НД05.02/01*)
	counterND050202: DWORD;		(*Счетчик включений НД05.02/02*)
	daysND050201: WORD;		(*Количество отработанных дней НД05.02/01*)
	hoursND050201: WORD;		(*Количество отработанных часов НД05.02/01*)
	minutesND050201: WORD;		(*Количество отработанных минут НД05.02/01*)
	secondsND050201: WORD;		(*Количество отработанных секунд НД05.02/01*)
	daysND050202: WORD;		(*Количество отработанных дней НД05.02/02*)
	hoursND050202: WORD;		(*Количество отработанных часов НД05.02/02*)
	minutesND050202: WORD;		(*Количество отработанных минут НД05.02/02*)
	secondsND050202: WORD;		(*Количество отработанных секунд НД05.02/02*)
	counterND060201: DWORD;		(*Счетчик включений НД06.02/01*)
	counterND060202: DWORD;		(*Счетчик включений НД06.02/02*)
	daysND060201: WORD;		(*Количество отработанных дней НД06.02/01*)
	hoursND060201: WORD;		(*Количество отработанных часов НД06.02/01*)
	minutesND060201: WORD;		(*Количество отработанных минут НД06.02/01*)
	secondsND060201: WORD;		(*Количество отработанных секунд НД06.02/01*)
	daysND060202: WORD;		(*Количество отработанных дней НД06.02/02*)
	hoursND060202: WORD;		(*Количество отработанных часов НД06.02/02*)
	minutesND060202: WORD;		(*Количество отработанных минут НД06.02/02*)
	secondsND060202: WORD;		(*Количество отработанных секунд НД06.02/02*)
	counterND060301: DWORD;		(*Счетчик включений НД06.03/01*)
	counterND060302: DWORD;		(*Счетчик включений НД06.03/02*)
	daysND060301: WORD;		(*Количество отработанных дней НД06.03/01*)
	hoursND060301: WORD;		(*Количество отработанных часов НД06.03/01*)
	minutesND060301: WORD;		(*Количество отработанных минут НД06.03/01*)
	secondsND060301: WORD;		(*Количество отработанных секунд НД06.03/01*)
	daysND060302: WORD;		(*Количество отработанных дней НД06.03/02*)
	hoursND060302: WORD;		(*Количество отработанных часов НД06.03/02*)
	minutesND060302: WORD;		(*Количество отработанных минут НД06.03/02*)
	secondsND060302: WORD;		(*Количество отработанных секунд НД06.03/02*)
	counterND070301: DWORD;		(*Счетчик включений НД07.03/01*)
	counterND070302: DWORD;		(*Счетчик включений НД07.03/02*)
	daysND070301: WORD;		(*Количество отработанных дней НД07.03/01*)
	hoursND070301: WORD;		(*Количество отработанных часов НД07.03/01*)
	minutesND070301: WORD;		(*Количество отработанных минут НД07.03/01*)
	secondsND070301: WORD;		(*Количество отработанных секунд НД07.03/01*)
	daysND070302: WORD;		(*Количество отработанных дней НД07.03/02*)
	hoursND070302: WORD;		(*Количество отработанных часов НД07.03/02*)
	minutesND070302: WORD;		(*Количество отработанных минут НД07.03/02*)
	secondsND070302: WORD;		(*Количество отработанных секунд НД07.03/02*)
	counterND080301: DWORD;		(*Счетчик включений НД08.03/01*)
	counterND080302: DWORD;		(*Счетчик включений НД08.03/02*)
	daysND080301: WORD;		(*Количество отработанных дней НД08.03/01*)
	hoursND080301: WORD;		(*Количество отработанных часов НД08.03/01*)
	minutesND080301: WORD;		(*Количество отработанных минут НД08.03/01*)
	secondsND080301: WORD;		(*Количество отработанных секунд НД08.03/01*)
	daysND080302: WORD;		(*Количество отработанных дней НД08.03/02*)
	hoursND080302: WORD;		(*Количество отработанных часов НД08.03/02*)
	minutesND080302: WORD;		(*Количество отработанных минут НД08.03/02*)
	secondsND080302: WORD;		(*Количество отработанных секунд НД08.03/02*)
	counterN010501: DWORD;		(*Счетчик включений Н01.05/01*)
	counterN010502: DWORD;		(*Счетчик включений Н01.05/02*)
	daysN010501: WORD;		(*Количество отработанных дней Н01.05/01*)
	hoursN010501: WORD;		(*Количество отработанных часов Н01.05/01*)
	minutesN010501: WORD;		(*Количество отработанных минут Н01.05/01*)
	secondsN010501: WORD;		(*Количество отработанных секунд Н01.05/01*)
	daysN010502: WORD;		(*Количество отработанных дней Н01.05/02*)
	hoursN010502: WORD;		(*Количество отработанных часов Н01.05/02*)
	minutesN010502: WORD;		(*Количество отработанных минут Н01.05/02*)
	secondsN010502: WORD;		(*Количество отработанных секунд Н01.05/02*)
	counterN020401: DWORD;		(*Счетчик включений Н02.04/01*)
	counterN020402: DWORD;		(*Счетчик включений Н02.04/02*)
	daysN020401: WORD;		(*Количество отработанных дней Н02.04/01*)
	hoursN020401: WORD;		(*Количество отработанных часов Н02.04/01*)
	minutesN020401: WORD;		(*Количество отработанных минут Н02.04/01*)
	secondsN020401: WORD;		(*Количество отработанных секунд Н02.04/01*)
	daysN020402: WORD;		(*Количество отработанных дней Н02.04/02*)
	hoursN020402: WORD;		(*Количество отработанных часов Н02.04/02*)
	minutesN020402: WORD;		(*Количество отработанных минут Н02.04/02*)
	secondsN020402: WORD;		(*Количество отработанных секунд Н02.04/02*)
	counterN040401: DWORD;		(*Счетчик включений Н04.04/01*)
	counterN040402: DWORD;		(*Счетчик включений Н04.04/02*)
	daysN040401: WORD;		(*Количество отработанных дней Н04.04/01*)
	hoursN040401: WORD;		(*Количество отработанных часов Н04.04/01*)
	minutesN040401: WORD;		(*Количество отработанных минут Н04.04/01*)
	secondsN040401: WORD;		(*Количество отработанных секунд Н04.04/01*)
	daysN040402: WORD;		(*Количество отработанных дней Н04.04/02*)
	hoursN040402: WORD;		(*Количество отработанных часов Н04.04/02*)
	minutesN040402: WORD;		(*Количество отработанных минут Н04.04/02*)
	secondsN040402: WORD;		(*Количество отработанных секунд Н04.04/02*)
	counterUFO030101: DWORD;		(*Счетчик включений УФО03.01/01*)
	counterUFO030102: DWORD;		(*Счетчик включений УФО03.01/02*)
	daysUFO030101: WORD;		(*Количество отработанных дней УФО03.01/01*)
	hoursUFO030101: WORD;		(*Количество отработанных часов УФО03.01/01*)
	minutesUFO030101: WORD;		(*Количество отработанных минут УФО03.01/01*)
	secondsUFO030101: WORD;		(*Количество отработанных секунд УФО03.01/01*)
	daysUFO030102: WORD;		(*Количество отработанных дней УФО03.01/02*)
	hoursUFO030102: WORD;		(*Количество отработанных часов УФО03.01/02*)
	minutesUFO030102: WORD;		(*Количество отработанных минут УФО03.01/02*)
	secondsUFO030102: WORD;		(*Количество отработанных секунд УФО03.01/02*)
END_VAR
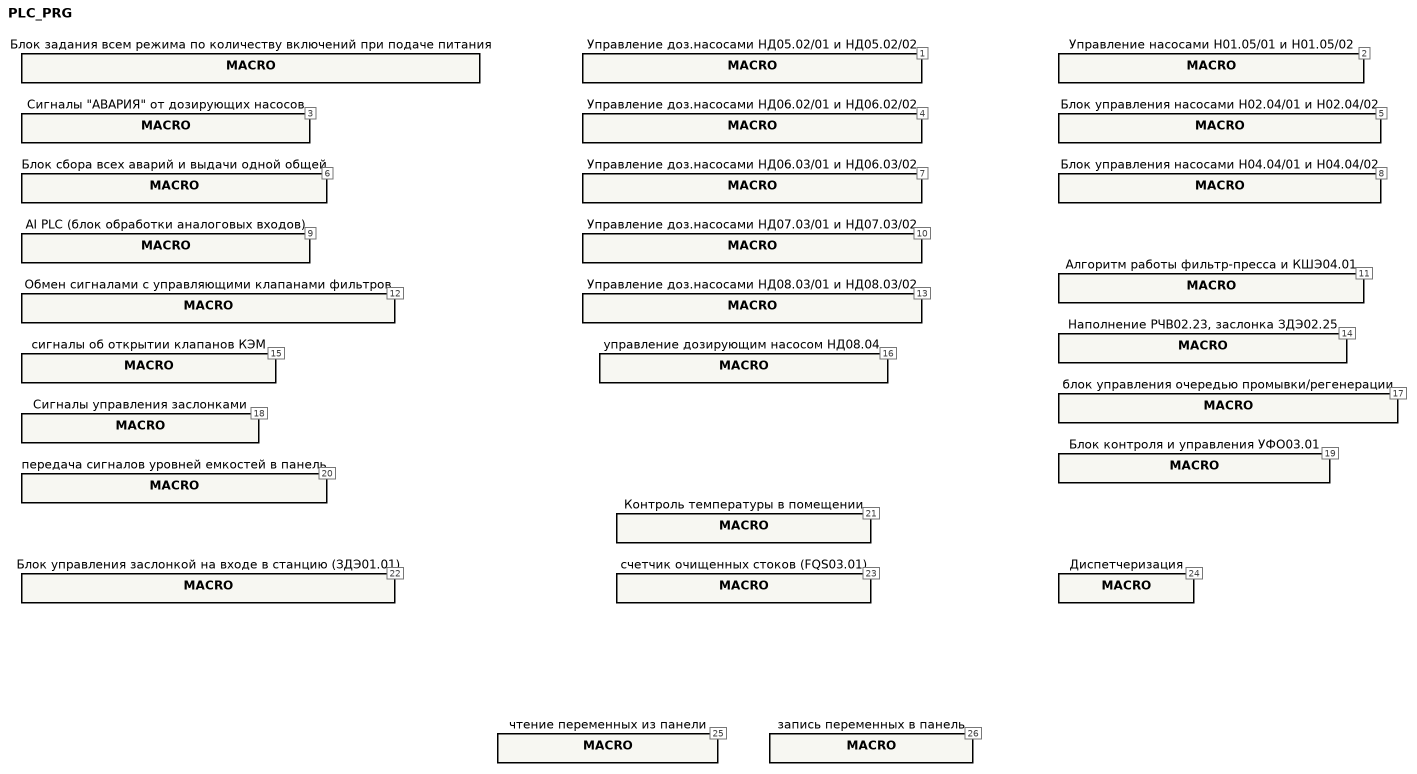
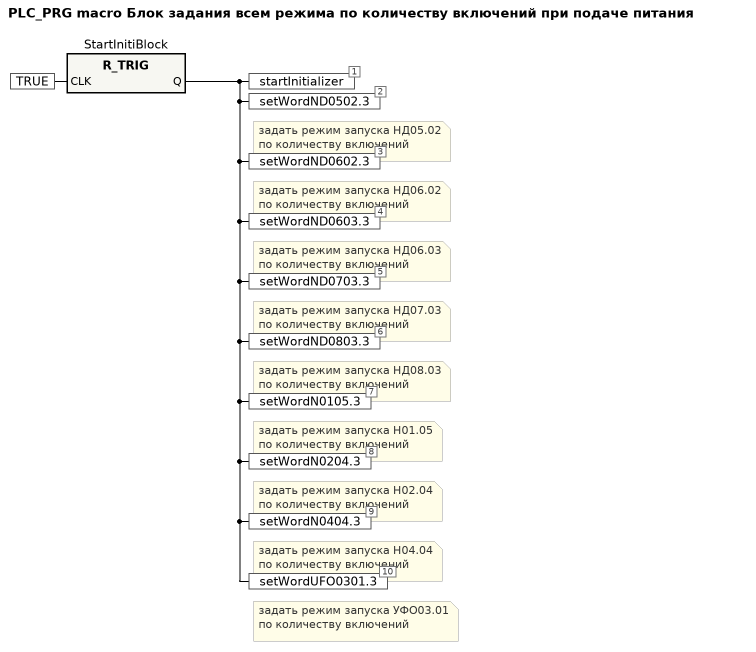
[picture p1: PLC_PRG macro Блок задания всем режима по количеству включений при подаче питания (CFC)]
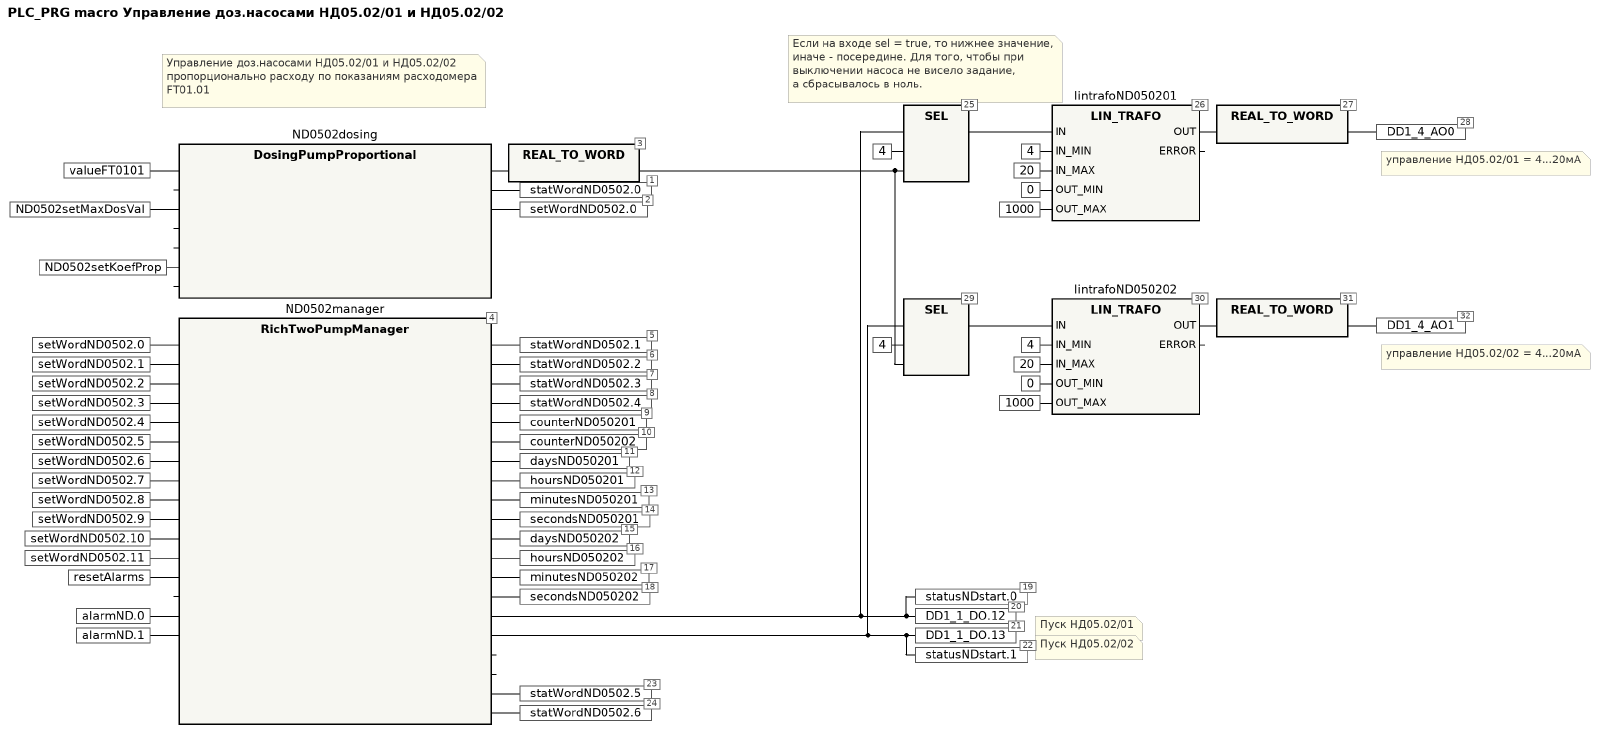
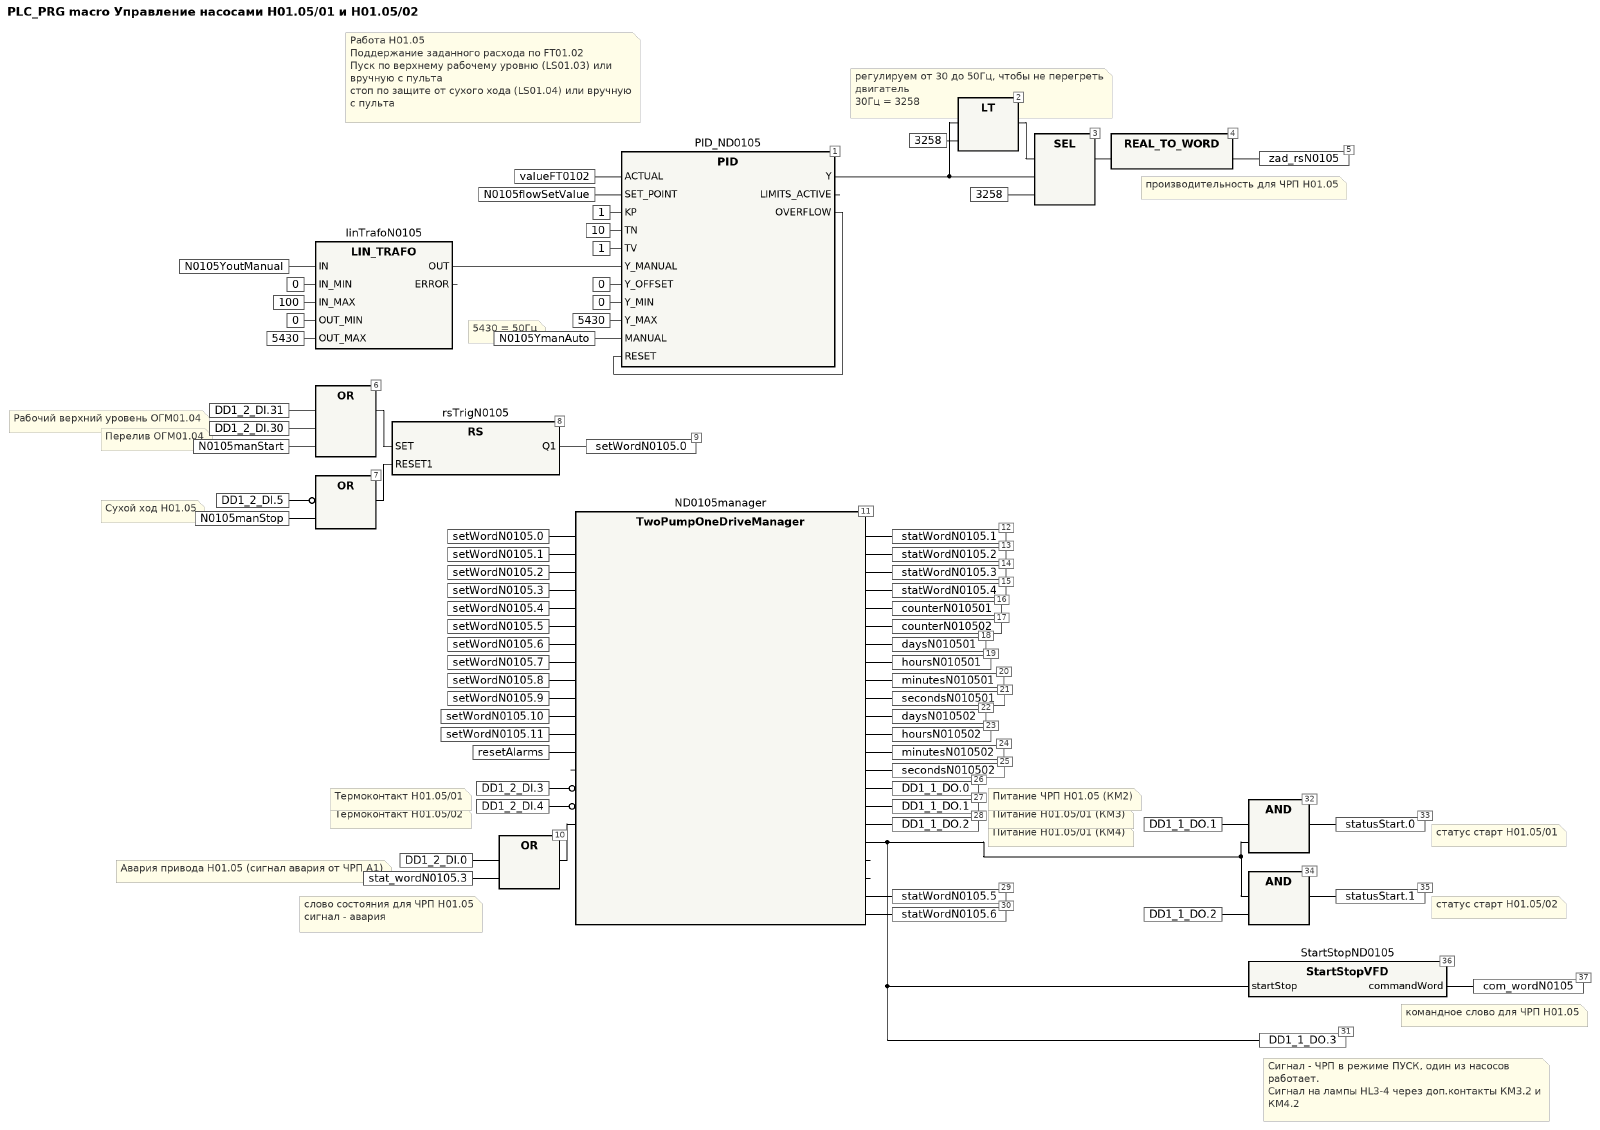
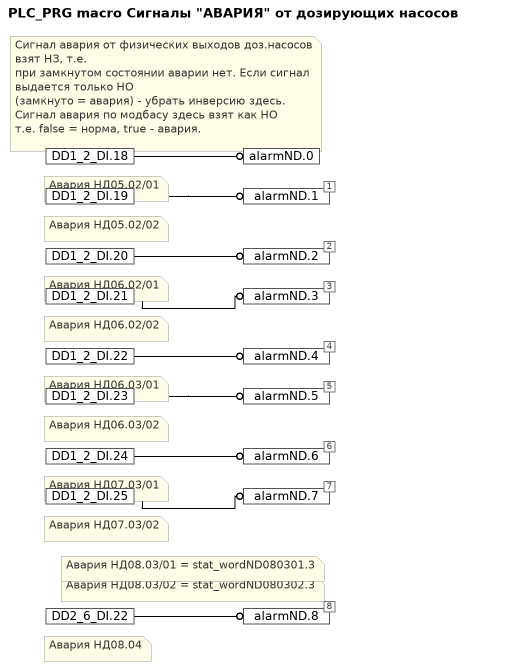
[picture p4: PLC_PRG macro Сигналы "АВАРИЯ" от дозирующих насосов (CFC)]
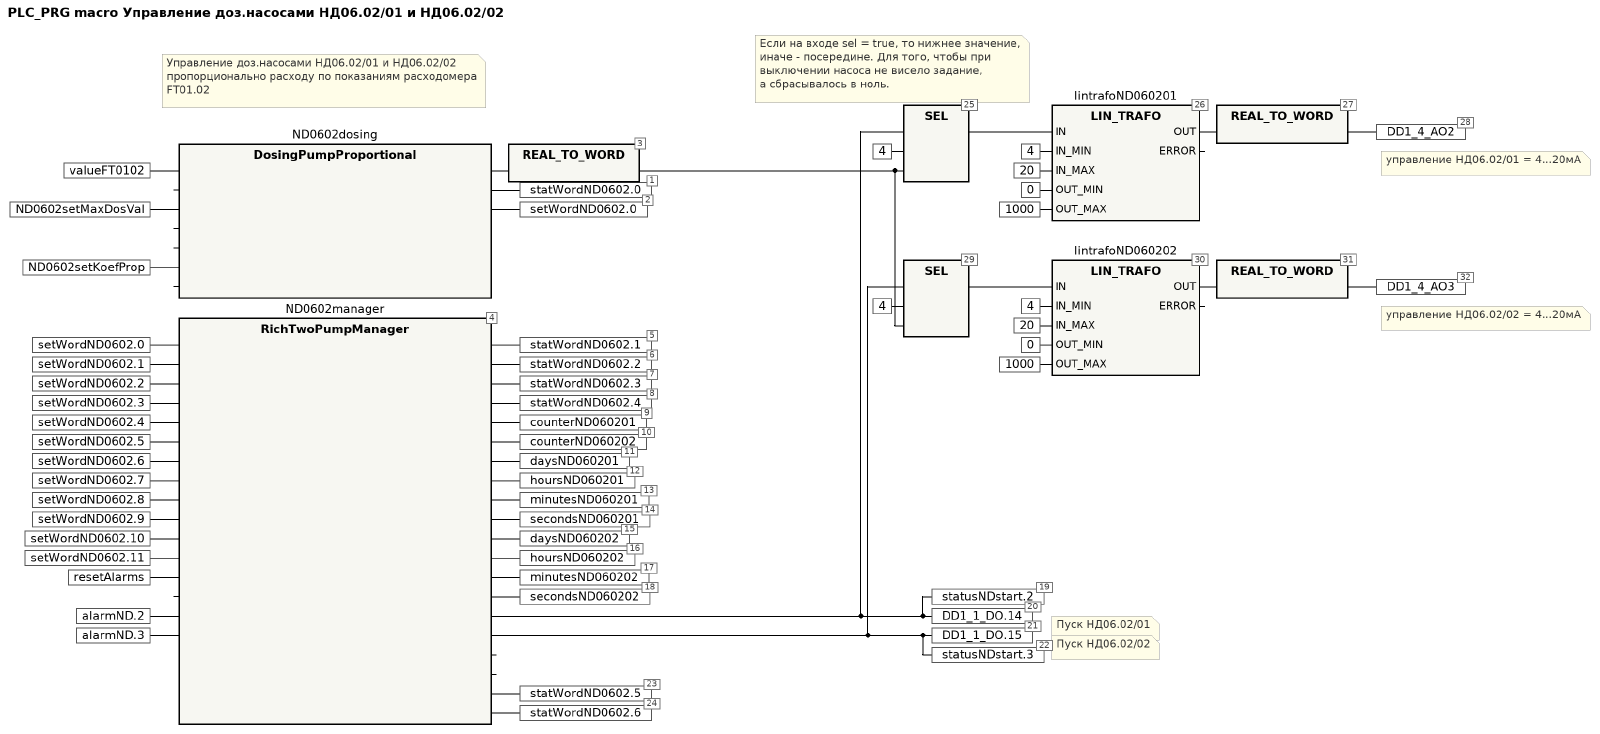
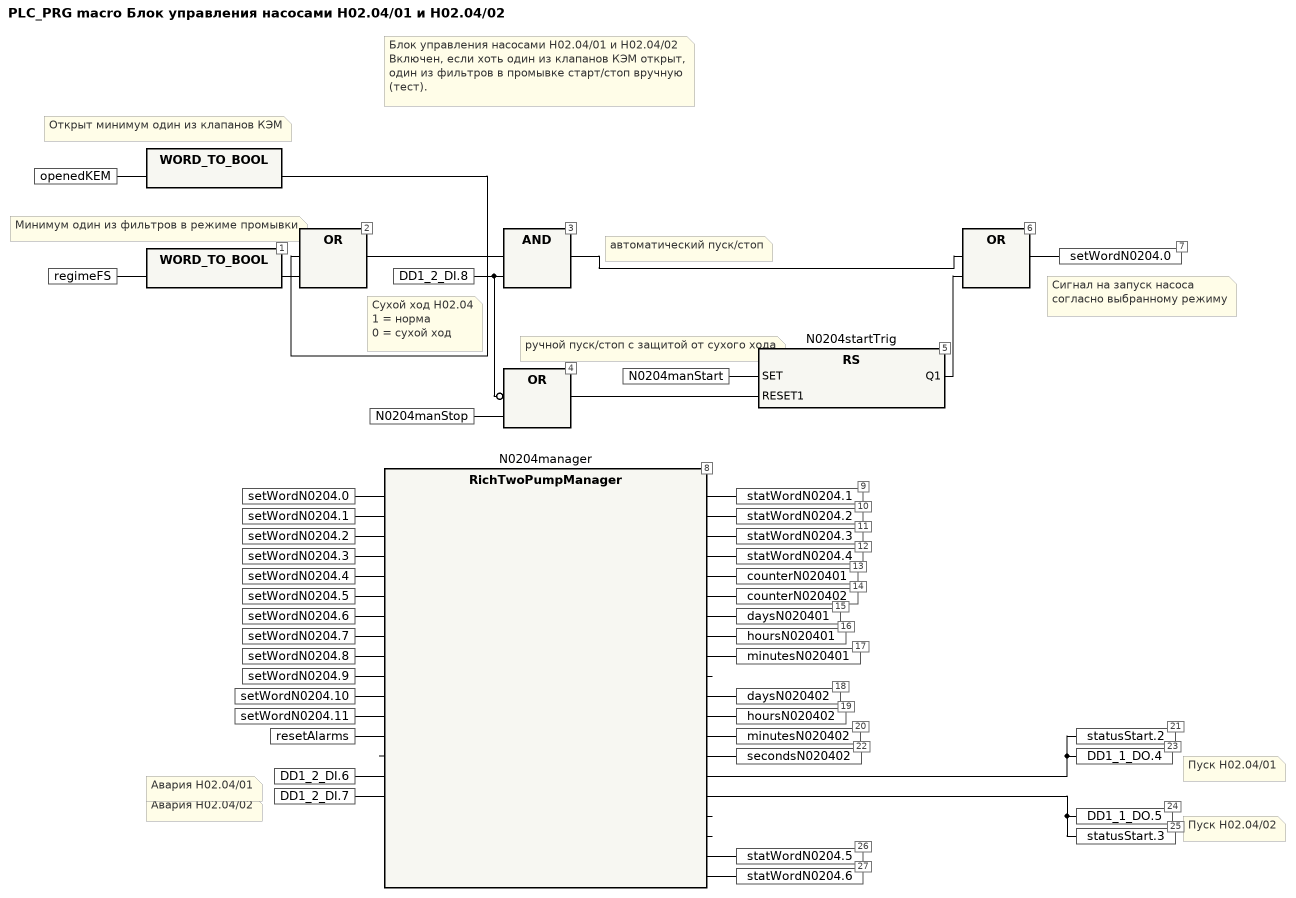
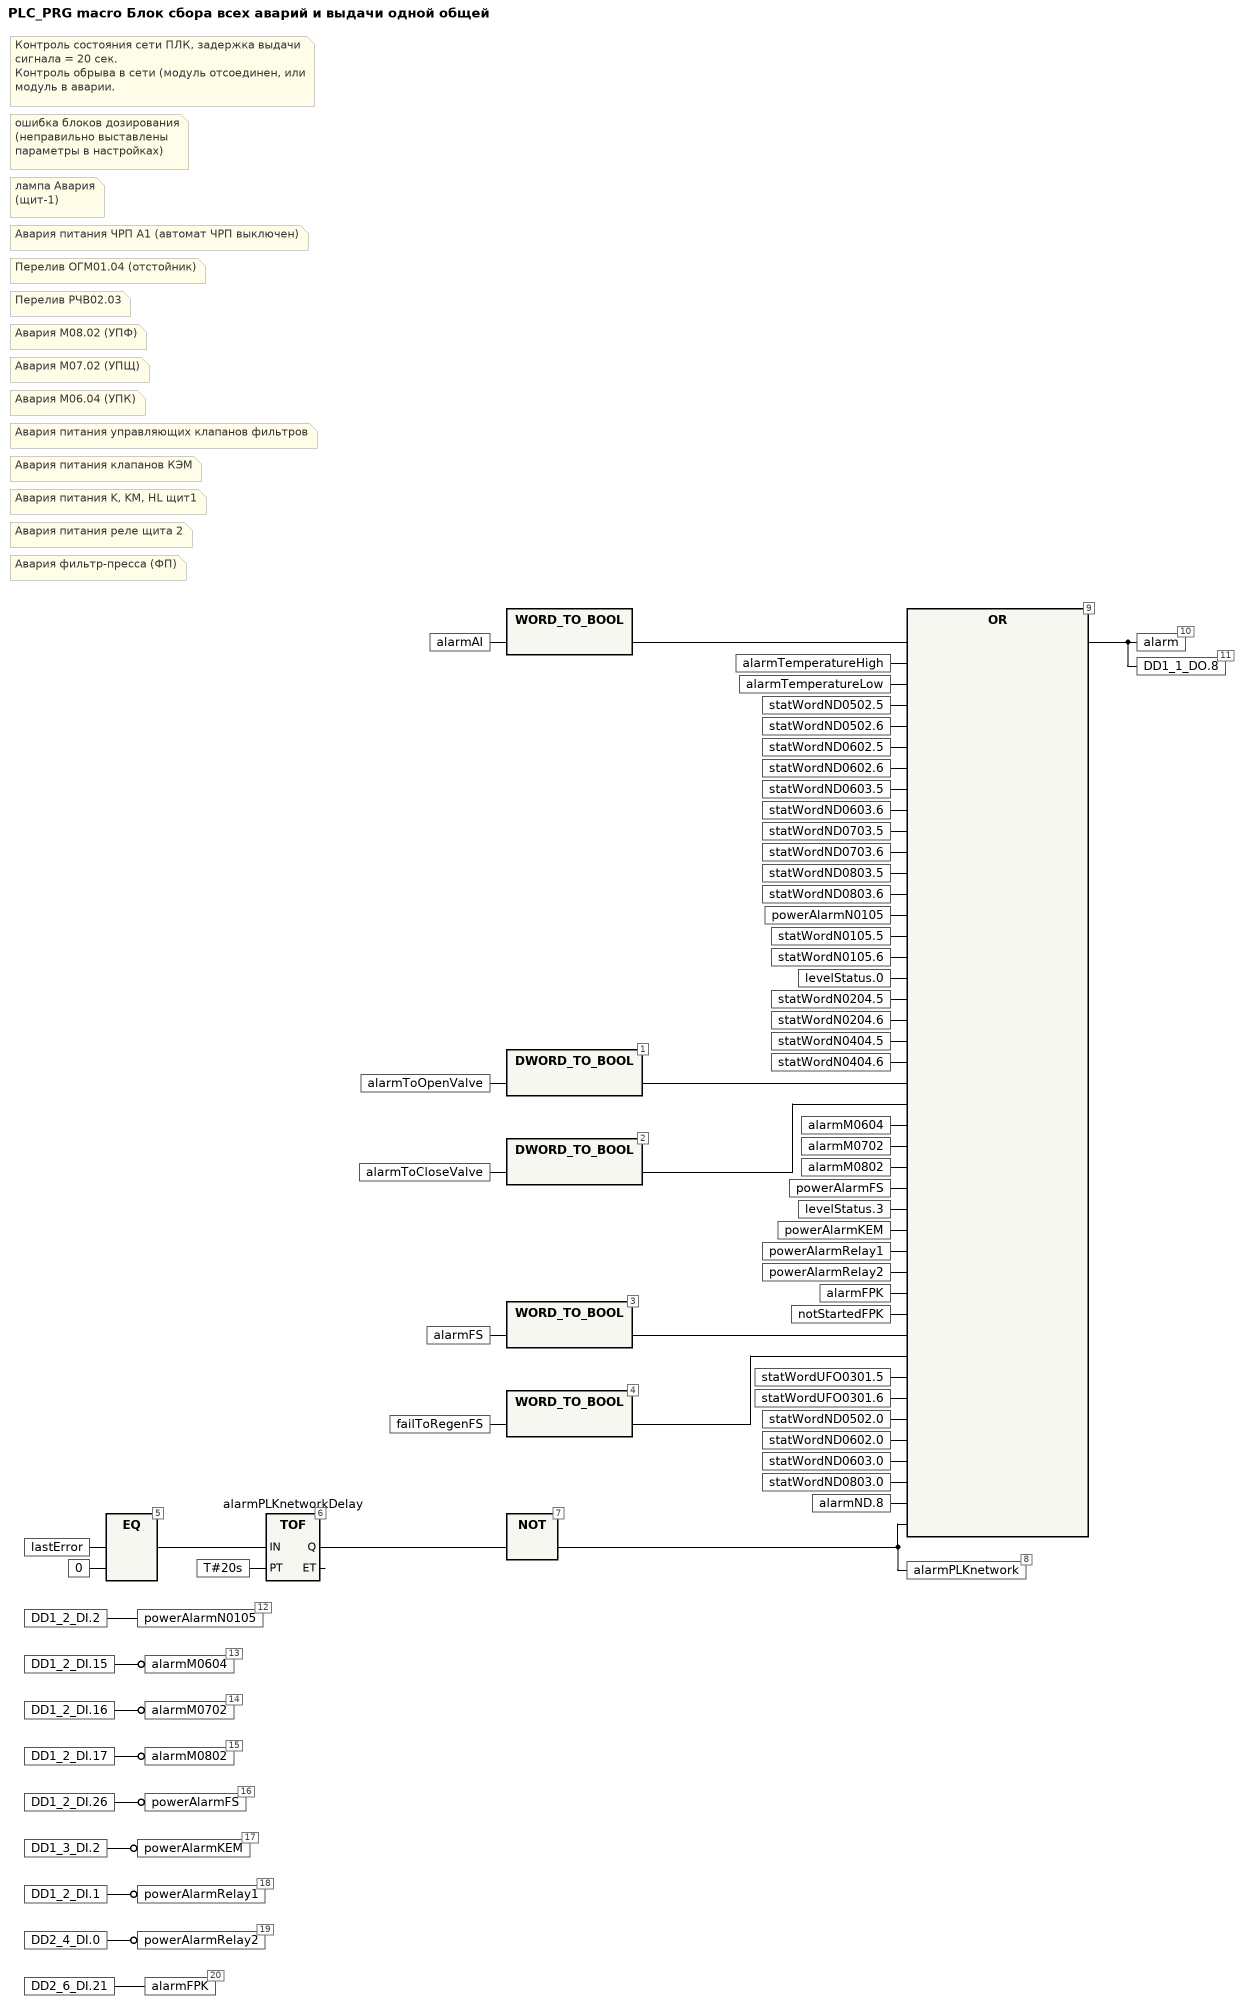
[picture p7: PLC_PRG macro Блок сбора всех аварий и выдачи одной общей (CFC)]
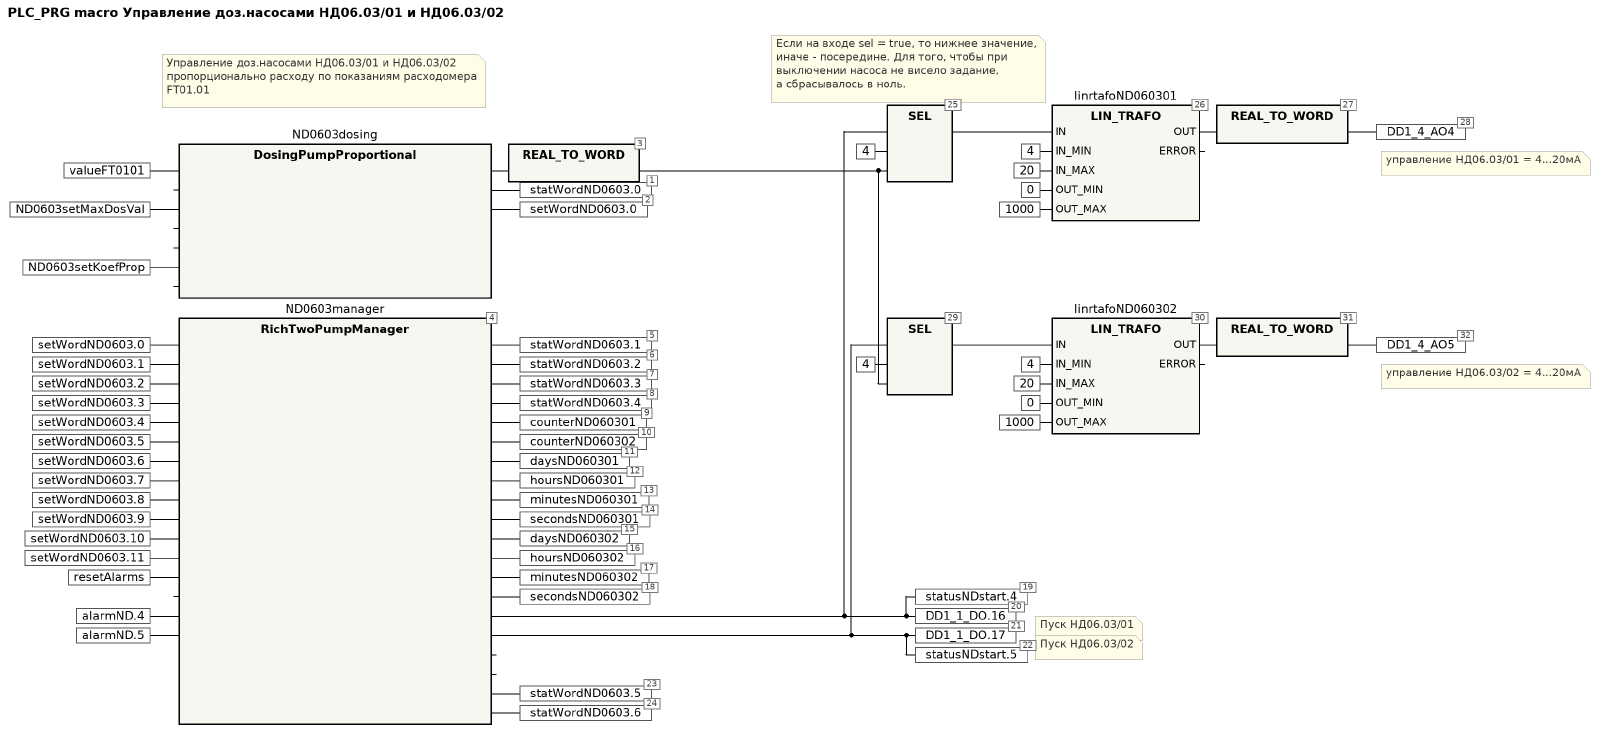
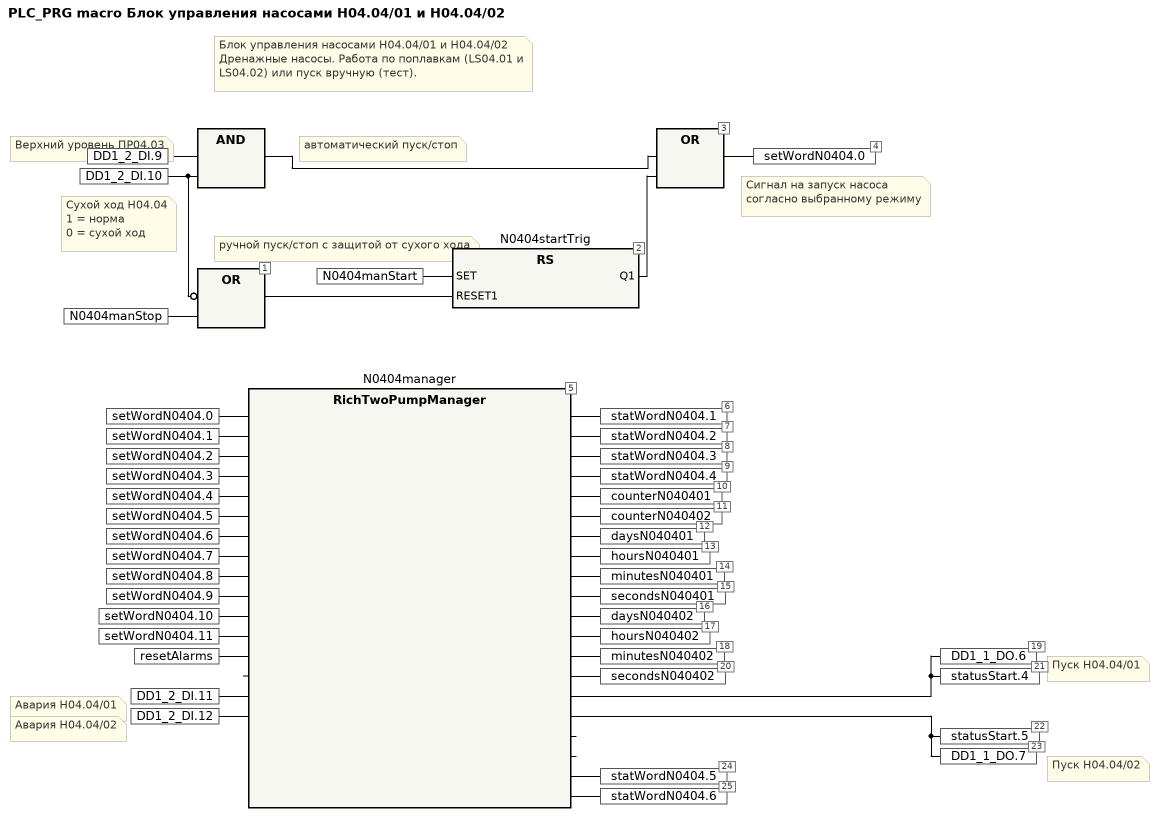
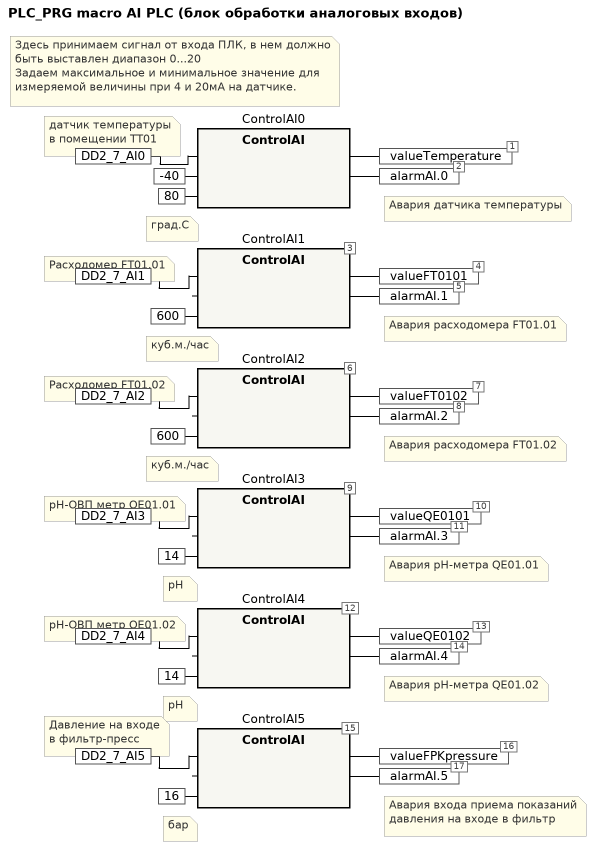
[picture p10: PLC_PRG macro AI PLC (блок обработки аналоговых входов) (CFC)]
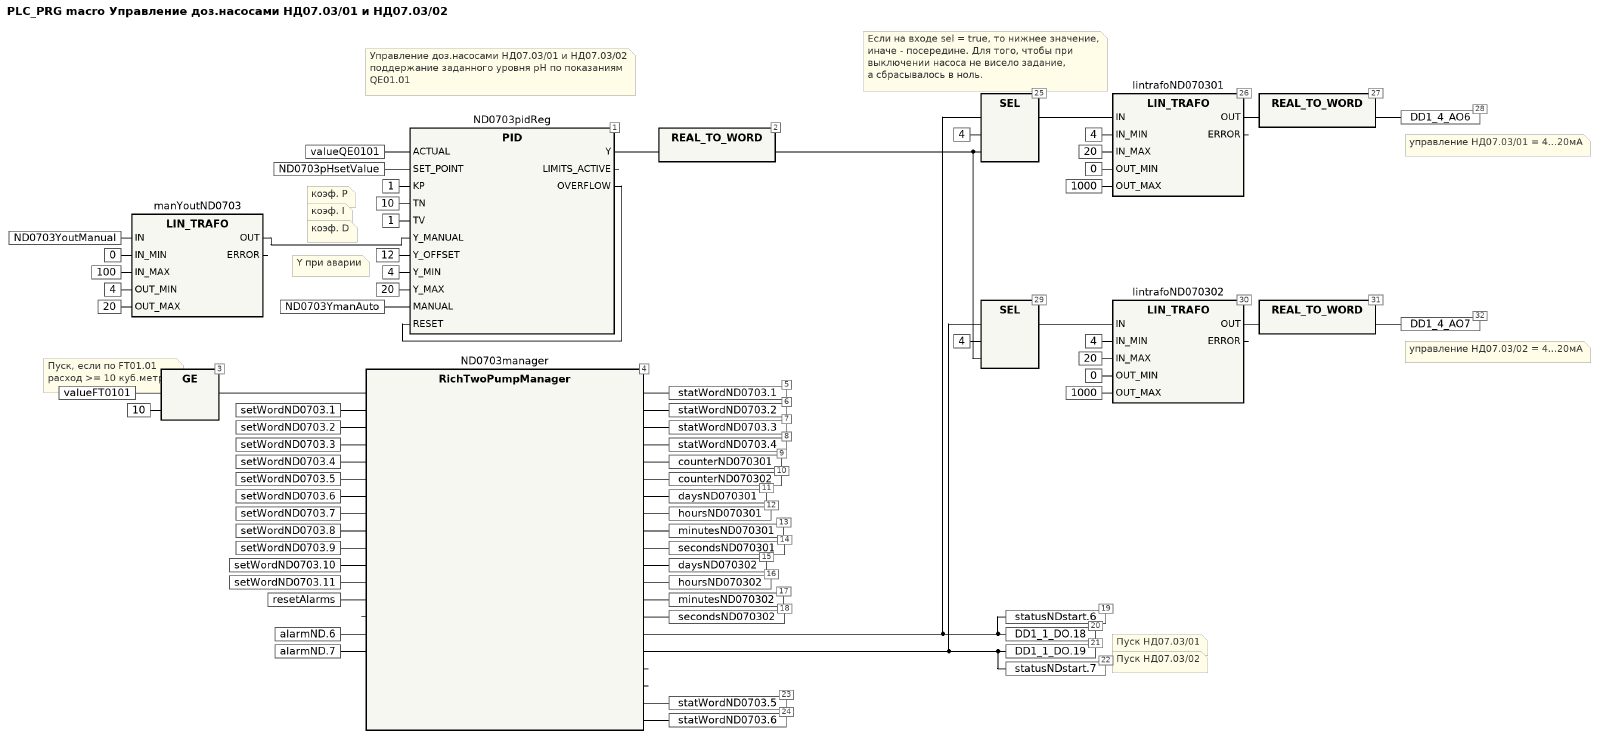
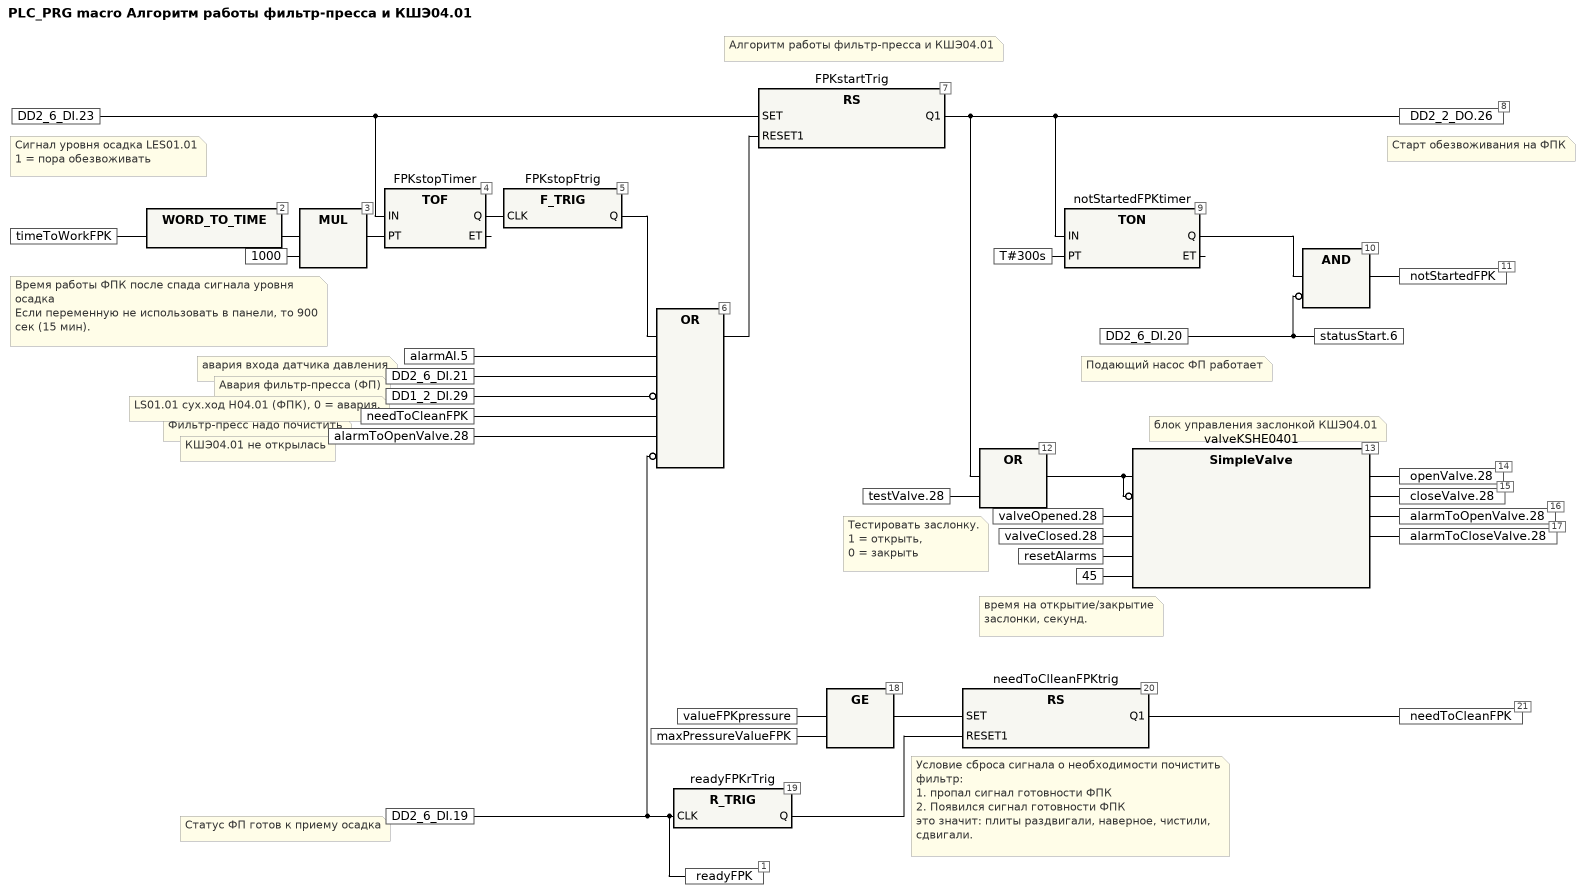
[picture p12: PLC_PRG macro Алгоритм работы фильтр-пресса и КШЭ04.01 (CFC)]
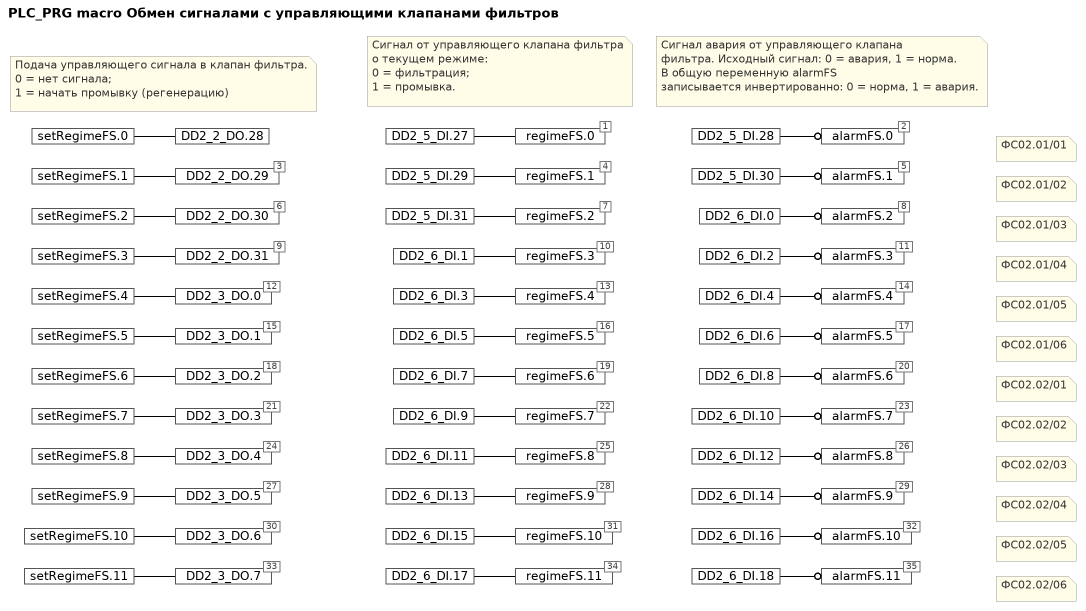
[picture p13: PLC_PRG macro Обмен сигналами с управляющими клапанами фильтров (CFC)]
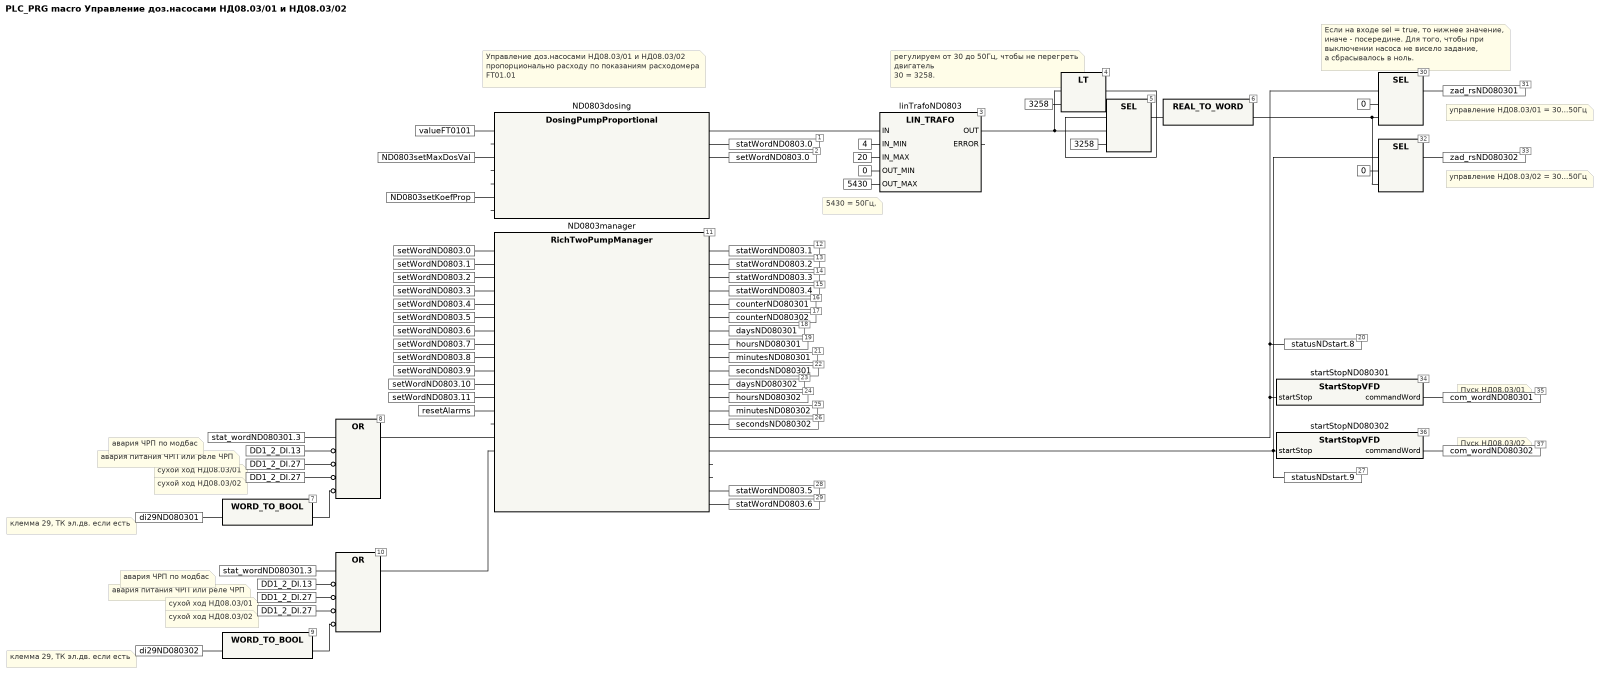
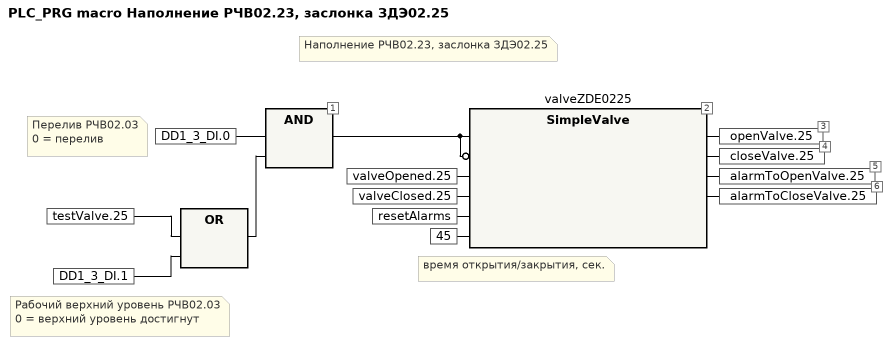
[picture p15: PLC_PRG macro Наполнение РЧВ02.23, заслонка ЗДЭ02.25 (CFC)]
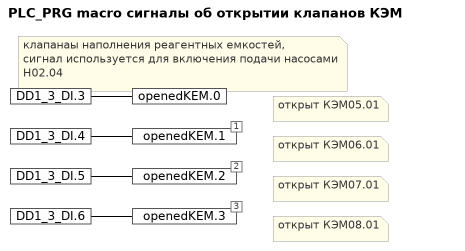
[picture p16: PLC_PRG macro сигналы об открытии клапанов КЭМ (CFC)]
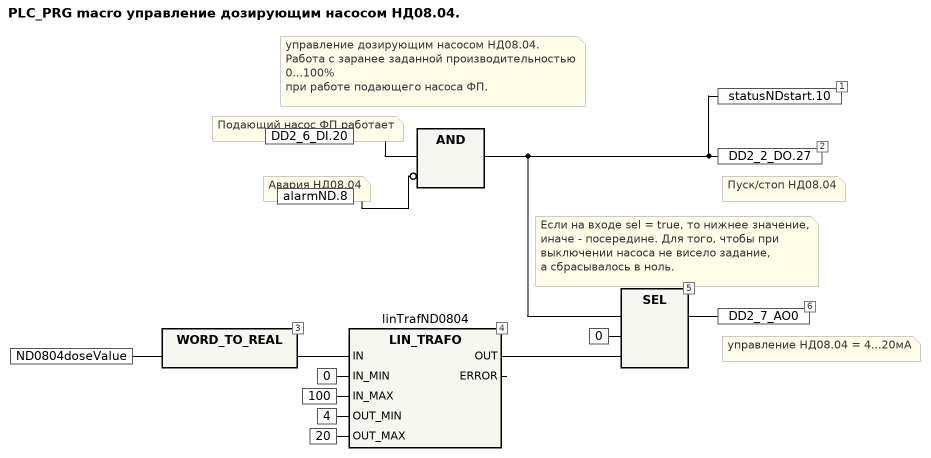
[picture p17: PLC_PRG macro управление дозирующим насосом НД08.04. (CFC)]
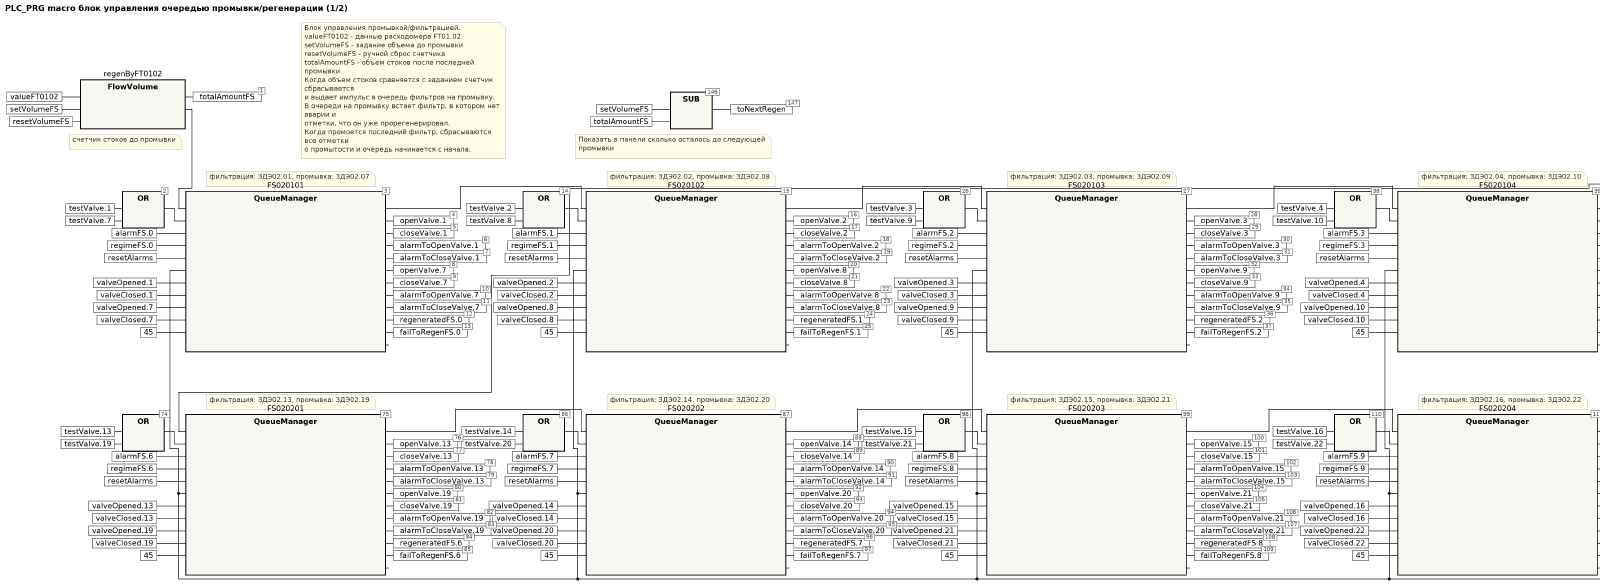
[picture p18: PLC_PRG macro блок управления очередью промывки/регенерации (CFC)]
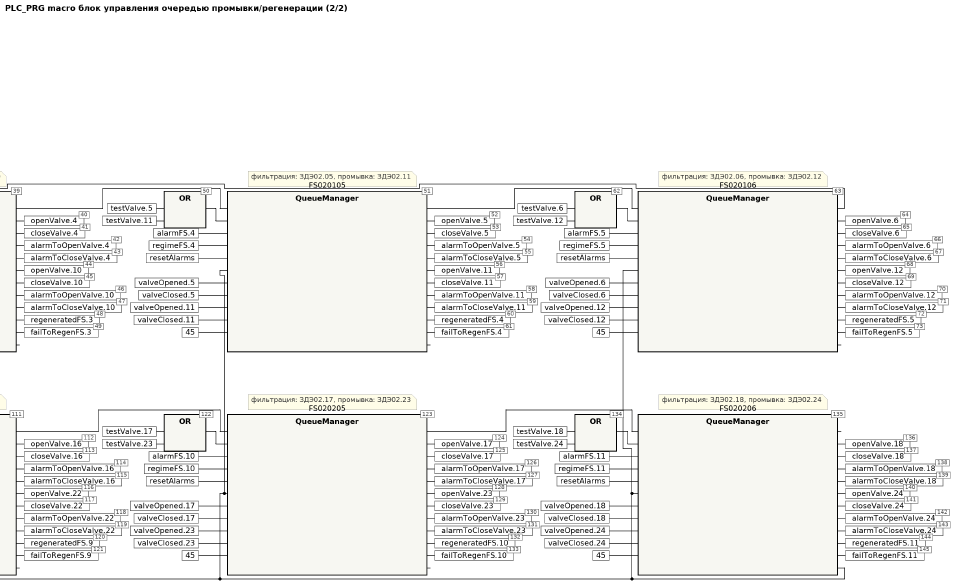
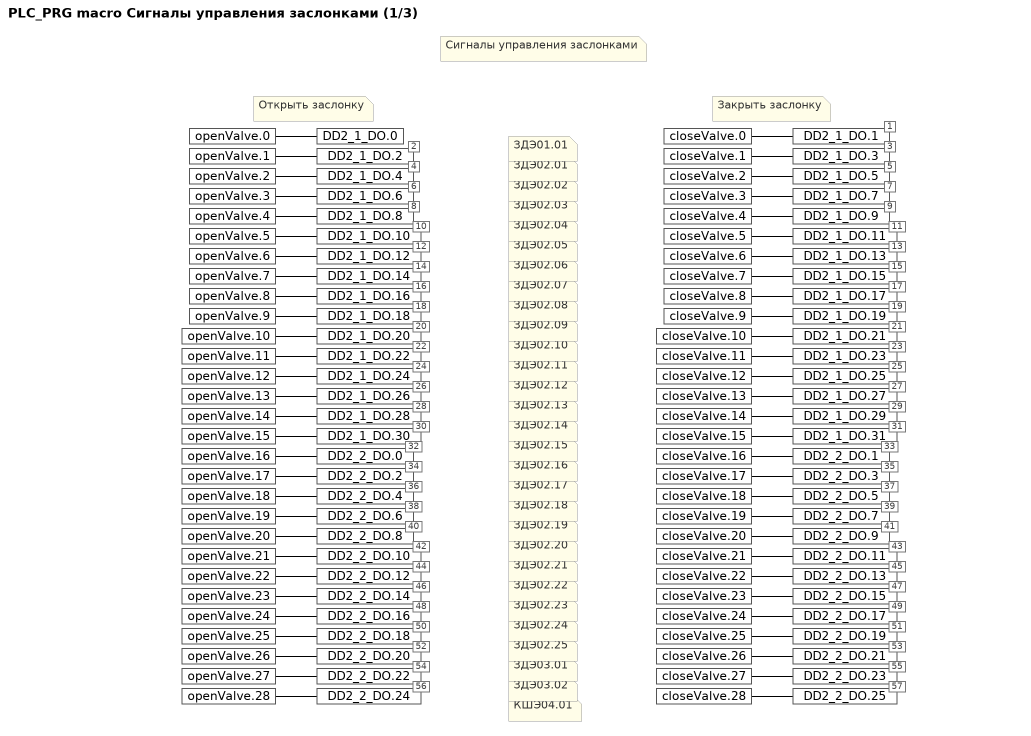
[picture p20: PLC_PRG macro Сигналы управления заслонками (CFC)]
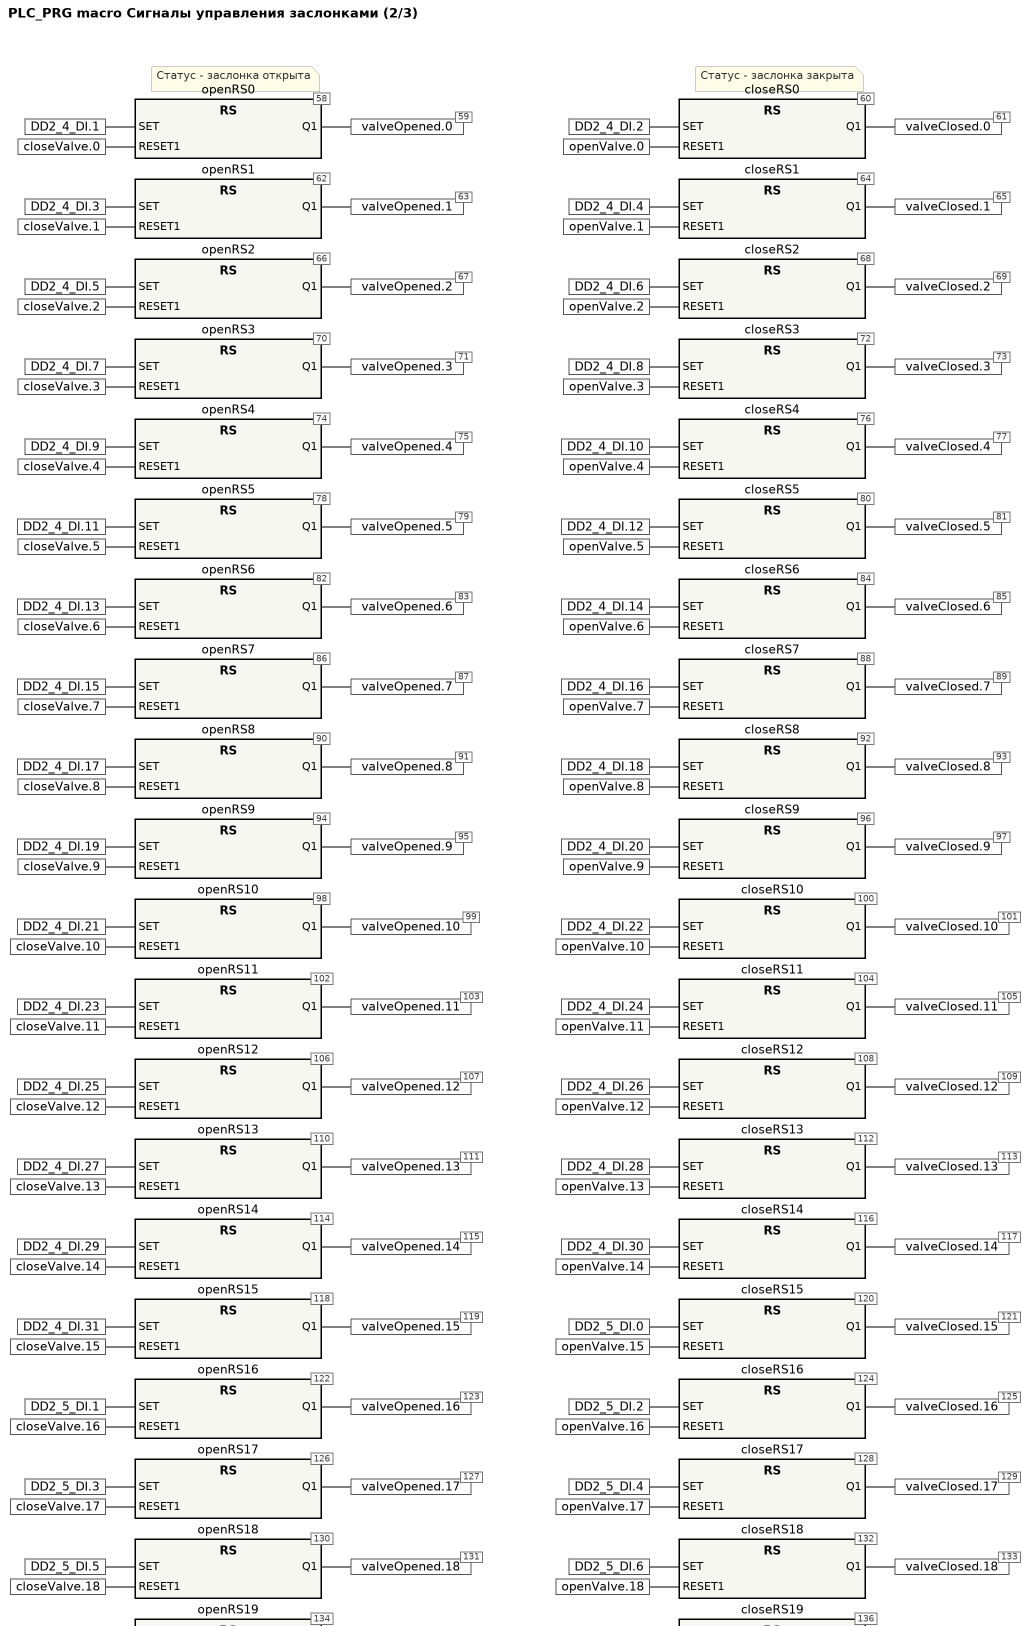
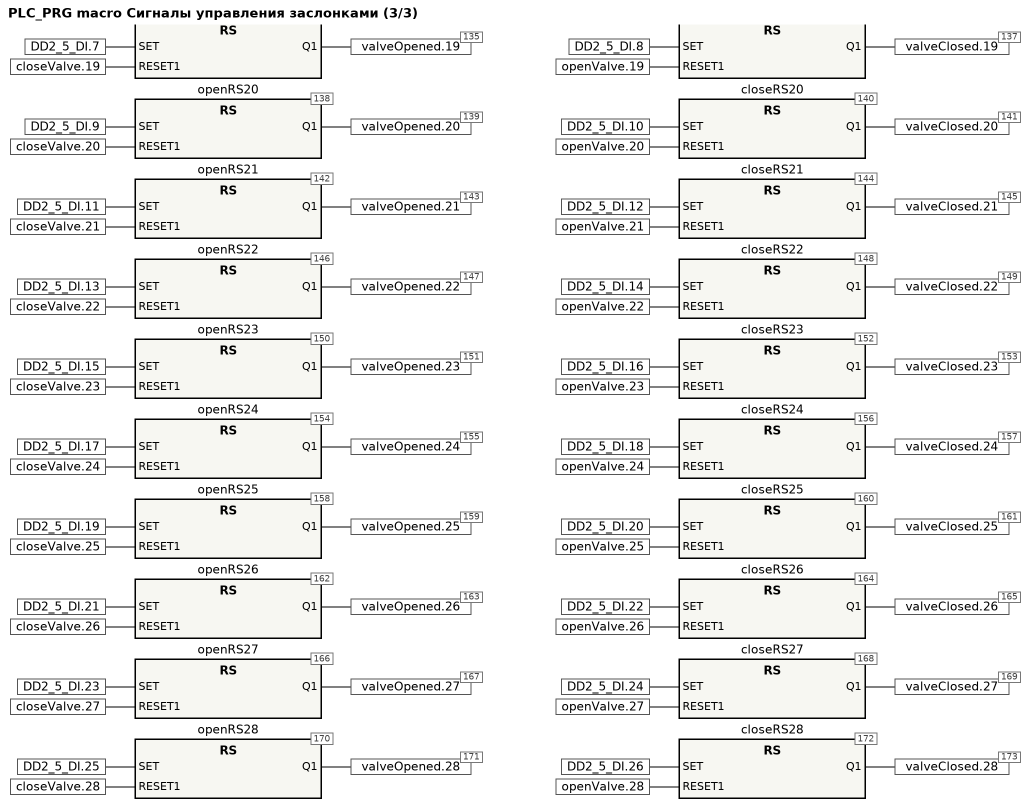
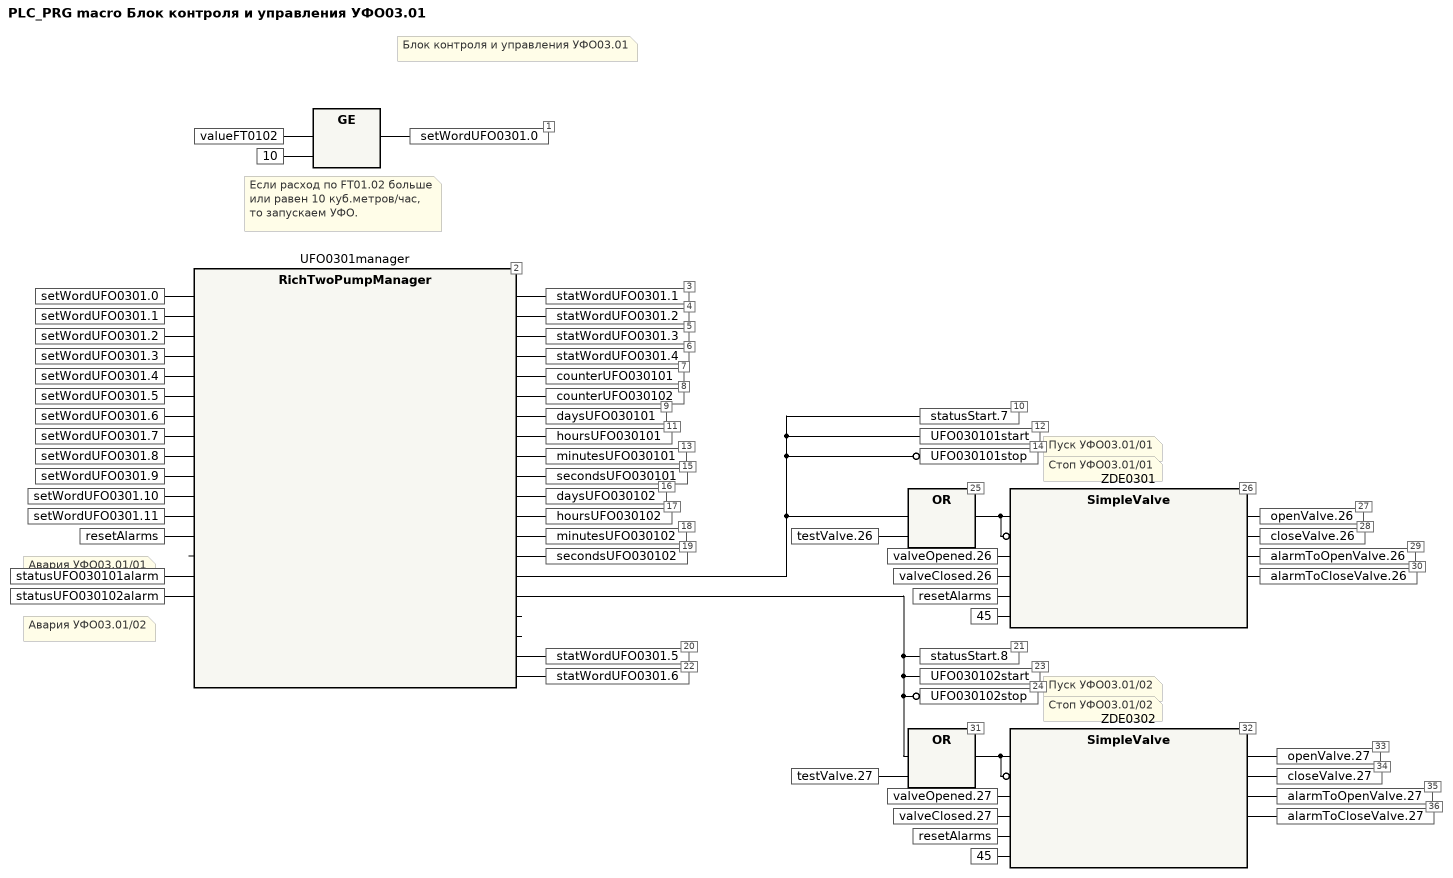
